REGION Network 65: Station 120 - Signalization (panel UH12)
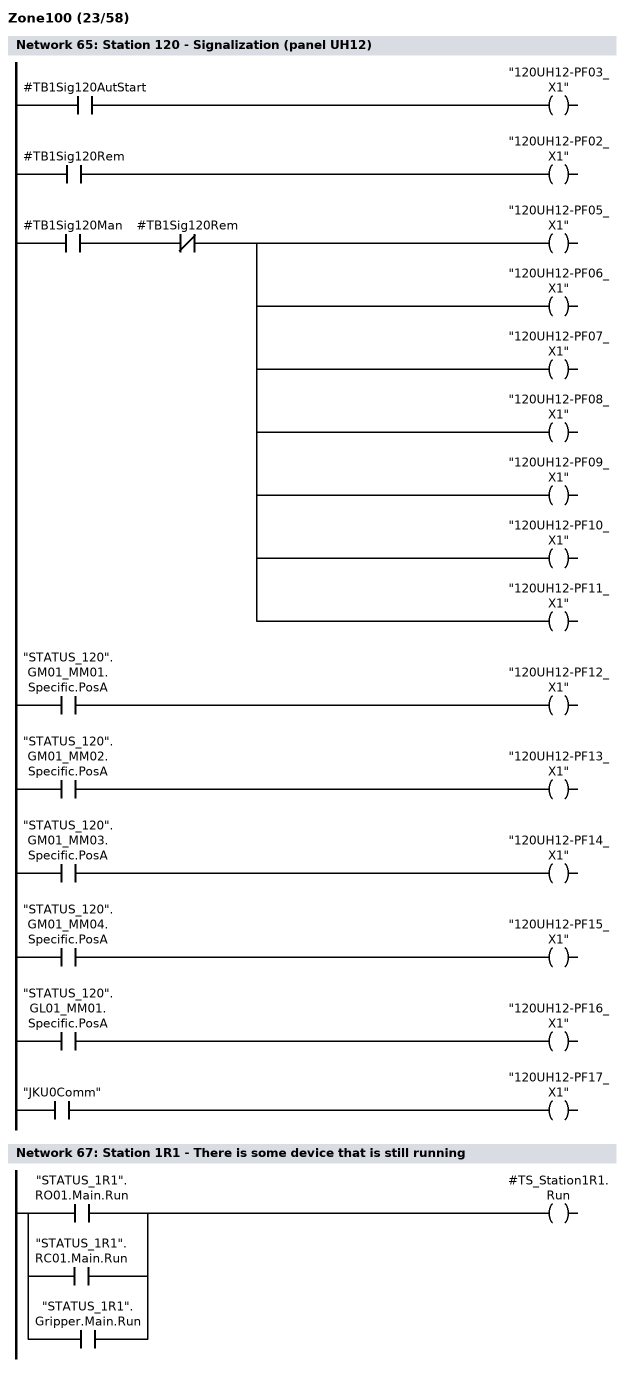
   RUNG wire#powerrail
      Contact( #TB1Sig120AutStart )
      Coil( "120UH12-PF03_X1" )
   END_RUNG
   RUNG wire#powerrail
      Contact( #TB1Sig120Rem )
      Coil( "120UH12-PF02_X1" )
   END_RUNG
   RUNG wire#powerrail
      Contact( #TB1Sig120Man )
      I_Contact( #TB1Sig120Rem )
      wire#w1
      Coil( "120UH12-PF05_X1" )
   END_RUNG
   RUNG wire#w1
      Coil( "120UH12-PF06_X1" )
   END_RUNG
   RUNG wire#w1
      Coil( "120UH12-PF07_X1" )
   END_RUNG
   RUNG wire#w1
      Coil( "120UH12-PF08_X1" )
   END_RUNG
   RUNG wire#w1
      Coil( "120UH12-PF09_X1" )
   END_RUNG
   RUNG wire#w1
      Coil( "120UH12-PF10_X1" )
   END_RUNG
   RUNG wire#w1
      Coil( "120UH12-PF11_X1" )
   END_RUNG
   RUNG wire#powerrail
      Contact( "STATUS_120".GM01_MM01.Specific.PosA )
      Coil( "120UH12-PF12_X1" )
   END_RUNG
   RUNG wire#powerrail
      Contact( "STATUS_120".GM01_MM02.Specific.PosA )
      Coil( "120UH12-PF13_X1" )
   END_RUNG
   RUNG wire#powerrail
      Contact( "STATUS_120".GM01_MM03.Specific.PosA )
      Coil( "120UH12-PF14_X1" )
   END_RUNG
   RUNG wire#powerrail
      Contact( "STATUS_120".GM01_MM04.Specific.PosA )
      Coil( "120UH12-PF15_X1" )
   END_RUNG
   RUNG wire#powerrail
      Contact( "STATUS_120".GL01_MM01.Specific.PosA )
      Coil( "120UH12-PF16_X1" )
   END_RUNG
   RUNG wire#powerrail
      Contact( "JKU0Comm" )
      Coil( "120UH12-PF17_X1" )
   END_RUNG
   // the same network as SCL:
   "120UH12-PF03_X1" := #TB1Sig120AutStart;
   "120UH12-PF02_X1" := #TB1Sig120Rem;
   "120UH12-PF05_X1" := #TB1Sig120Man AND NOT #TB1Sig120Rem;
   "120UH12-PF06_X1" := "120UH12-PF05_X1";
   "120UH12-PF07_X1" := "120UH12-PF05_X1";
   "120UH12-PF08_X1" := "120UH12-PF05_X1";
   "120UH12-PF09_X1" := "120UH12-PF05_X1";
   "120UH12-PF10_X1" := "120UH12-PF05_X1";
   "120UH12-PF11_X1" := "120UH12-PF05_X1";
   "120UH12-PF12_X1" := "STATUS_120".GM01_MM01.Specific.PosA;
   "120UH12-PF13_X1" := "STATUS_120".GM01_MM02.Specific.PosA;
   "120UH12-PF14_X1" := "STATUS_120".GM01_MM03.Specific.PosA;
   "120UH12-PF15_X1" := "STATUS_120".GM01_MM04.Specific.PosA;
   "120UH12-PF16_X1" := "STATUS_120".GL01_MM01.Specific.PosA;
   "120UH12-PF17_X1" := "JKU0Comm";
END_REGION

REGION Network 66: *************** Station 1R1 ***************
END_REGION

REGION Network 67: Station 1R1 - There is some device that is still running
   RUNG wire#powerrail
      Contact( "STATUS_1R1".RO01.Main.Run )
      wire#w1
      Coil( #TS_Station1R1.Run )
   END_RUNG
   RUNG wire#powerrail
      Contact( "STATUS_1R1".RC01.Main.Run )
   END_RUNG wire#w1
   RUNG wire#powerrail
      Contact( "STATUS_1R1".Gripper.Main.Run )
   END_RUNG wire#w1
   // the same network as SCL:
   #TS_Station1R1.Run := "STATUS_1R1".RO01.Main.Run OR "STATUS_1R1".RC01.Main.Run OR "STATUS_1R1".Gripper.Main.Run;
END_REGION

REGION Network 68: Station 1R1 - Warning
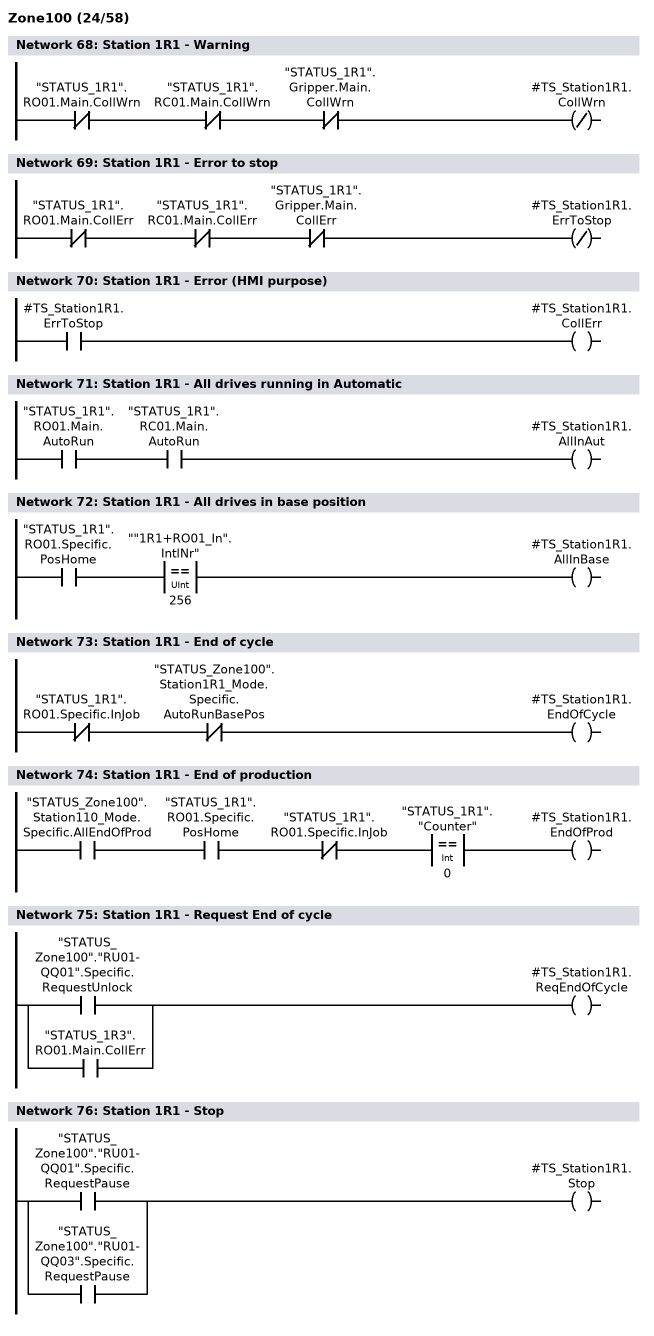
   RUNG wire#powerrail
      I_Contact( "STATUS_1R1".RO01.Main.CollWrn )
      I_Contact( "STATUS_1R1".RC01.Main.CollWrn )
      I_Contact( "STATUS_1R1".Gripper.Main.CollWrn )
      I_Coil( #TS_Station1R1.CollWrn )
   END_RUNG
   // the same network as SCL:
   #TS_Station1R1.CollWrn := NOT (NOT "STATUS_1R1".RO01.Main.CollWrn AND NOT "STATUS_1R1".RC01.Main.CollWrn AND NOT "STATUS_1R1".Gripper.Main.CollWrn);
END_REGION

REGION Network 69: Station 1R1 - Error to stop
   RUNG wire#powerrail
      I_Contact( "STATUS_1R1".RO01.Main.CollErr )
      I_Contact( "STATUS_1R1".RC01.Main.CollErr )
      I_Contact( "STATUS_1R1".Gripper.Main.CollErr )
      I_Coil( #TS_Station1R1.ErrToStop )
   END_RUNG
   // the same network as SCL:
   #TS_Station1R1.ErrToStop := NOT (NOT "STATUS_1R1".RO01.Main.CollErr AND NOT "STATUS_1R1".RC01.Main.CollErr AND NOT "STATUS_1R1".Gripper.Main.CollErr);
END_REGION

REGION Network 70: Station 1R1 - Error (HMI purpose)
   RUNG wire#powerrail
      Contact( #TS_Station1R1.ErrToStop )
      Coil( #TS_Station1R1.CollErr )
   END_RUNG
   // the same network as SCL:
   #TS_Station1R1.CollErr := #TS_Station1R1.ErrToStop;
END_REGION

REGION Network 71: Station 1R1 - All drives running in Automatic
   RUNG wire#powerrail
      Contact( "STATUS_1R1".RO01.Main.AutoRun )
      Contact( "STATUS_1R1".RC01.Main.AutoRun )
      Coil( #TS_Station1R1.AllInAut )
   END_RUNG
   // the same network as SCL:
   #TS_Station1R1.AllInAut := "STATUS_1R1".RO01.Main.AutoRun AND "STATUS_1R1".RC01.Main.AutoRun;
END_REGION

REGION Network 72: Station 1R1 - All drives in base position
   RUNG wire#powerrail
      Contact( "STATUS_1R1".RO01.Specific.PosHome )
      { S7_Templates := "SrcType := UInt" } EQ_Contact(in1 := ""1R1+RO01_In".IntlNr", in2 := 256)
      Coil( #TS_Station1R1.AllInBase )
   END_RUNG
   // the same network as SCL:
   // no checked SCL form for this network; see the picture
END_REGION

REGION Network 73: Station 1R1 - End of cycle
   RUNG wire#powerrail
      I_Contact( "STATUS_1R1".RO01.Specific.InJob )
      I_Contact( "STATUS_Zone100".Station1R1_Mode.Specific.AutoRunBasePos )
      Coil( #TS_Station1R1.EndOfCycle )
   END_RUNG
   // the same network as SCL:
   #TS_Station1R1.EndOfCycle := NOT "STATUS_1R1".RO01.Specific.InJob AND NOT "STATUS_Zone100".Station1R1_Mode.Specific.AutoRunBasePos;
END_REGION

REGION Network 74: Station 1R1 - End of production
   RUNG wire#powerrail
      Contact( "STATUS_Zone100".Station110_Mode.Specific.AllEndOfProd )
      Contact( "STATUS_1R1".RO01.Specific.PosHome )
      I_Contact( "STATUS_1R1".RO01.Specific.InJob )
      { S7_Templates := "SrcType := Int" } EQ_Contact(in1 := "STATUS_1R1"."Counter", in2 := 0)
      Coil( #TS_Station1R1.EndOfProd )
   END_RUNG
   // the same network as SCL:
   #TS_Station1R1.EndOfProd := "STATUS_Zone100".Station110_Mode.Specific.AllEndOfProd AND "STATUS_1R1".RO01.Specific.PosHome AND NOT "STATUS_1R1".RO01.Specific.InJob AND ("STATUS_1R1"."Counter" = 0);
END_REGION

REGION Network 75: Station 1R1 - Request End of cycle
   RUNG wire#powerrail
      Contact( "STATUS_Zone100"."RU01-QQ01".Specific.RequestUnlock )
      wire#w1
      Coil( #TS_Station1R1.ReqEndOfCycle )
   END_RUNG
   RUNG wire#powerrail
      Contact( "STATUS_1R3".RO01.Main.CollErr )
   END_RUNG wire#w1
   // the same network as SCL:
   #TS_Station1R1.ReqEndOfCycle := "STATUS_Zone100"."RU01-QQ01".Specific.RequestUnlock OR "STATUS_1R3".RO01.Main.CollErr;
END_REGION

REGION Network 76: Station 1R1 - Stop
   RUNG wire#powerrail
      Contact( "STATUS_Zone100"."RU01-QQ01".Specific.RequestPause )
      wire#w1
      Coil( #TS_Station1R1.Stop )
   END_RUNG
   RUNG wire#powerrail
      Contact( "STATUS_Zone100"."RU01-QQ03".Specific.RequestPause )
   END_RUNG wire#w1
   // the same network as SCL:
   #TS_Station1R1.Stop := "STATUS_Zone100"."RU01-QQ01".Specific.RequestPause OR "STATUS_Zone100"."RU01-QQ03".Specific.RequestPause;
END_REGION

REGION Network 77: Station 1R1 - Number of selected devices
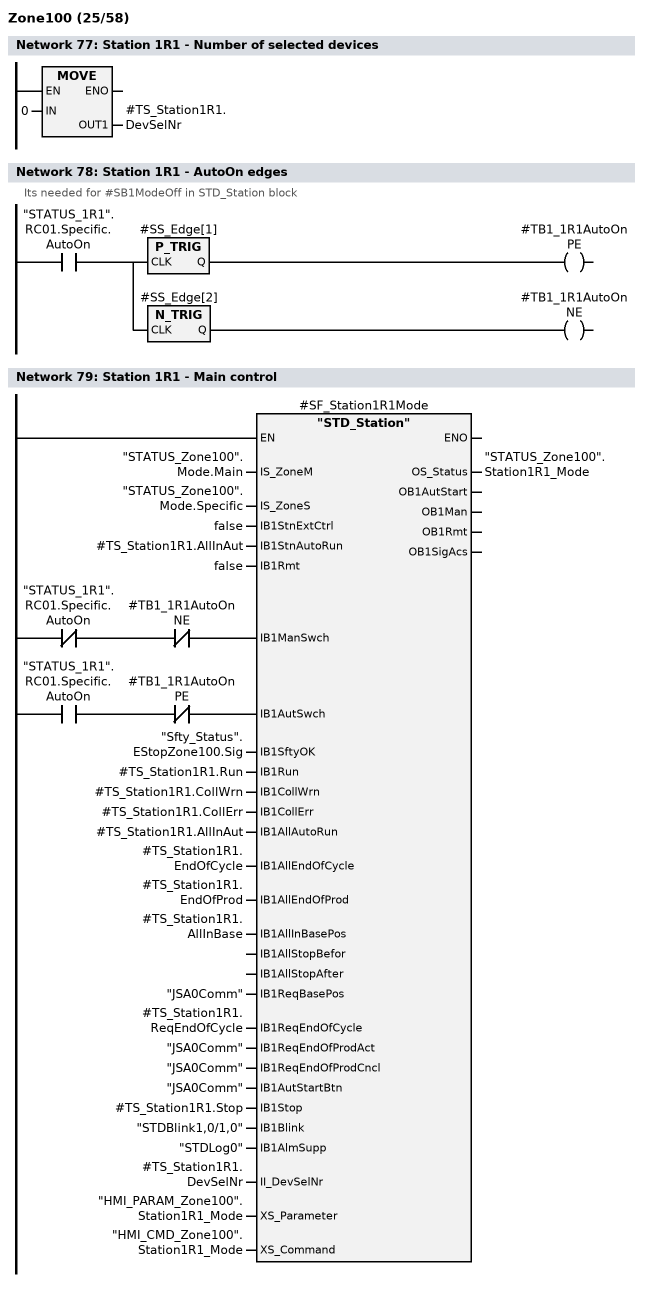
   RUNG wire#powerrail
      Move(in := 0, out1 => #TS_Station1R1.DevSelNr)
   END_RUNG
   // the same network as SCL:
   #TS_Station1R1.DevSelNr := 0;
END_REGION

REGION Network 78: Station 1R1 - AutoOn edges
   // Its needed for #SB1ModeOff in STD_Station block
   RUNG wire#powerrail
      Contact( "STATUS_1R1".RC01.Specific.AutoOn )
      wire#w1
      P_Trig( #SS_Edge[1] )
      Coil( #TB1_1R1AutoOnPE )
   END_RUNG
   RUNG wire#w1
      N_Trig( #SS_Edge[2] )
      Coil( #TB1_1R1AutoOnNE )
   END_RUNG
   // the same network as SCL:
   #_w1 := "STATUS_1R1".RC01.Specific.AutoOn AND NOT #SS_Edge[1];   // rising edge
   #SS_Edge[1] := "STATUS_1R1".RC01.Specific.AutoOn;
   #TB1_1R1AutoOnPE := #_w1;
   #_w2 := NOT "STATUS_1R1".RC01.Specific.AutoOn AND #SS_Edge[2];   // falling edge
   #SS_Edge[2] := "STATUS_1R1".RC01.Specific.AutoOn;
   #TB1_1R1AutoOnNE := #_w2;
END_REGION

REGION Network 79: Station 1R1 - Main control
   RUNG wire#powerrail
      #SF_Station1R1Mode(IB1ManSwch := wire#w1, IB1AutSwch := wire#w2, IS_ZoneM := "STATUS_Zone100".Mode.Main, IS_ZoneS := "STATUS_Zone100".Mode.Specific, IB1StnExtCtrl := false, IB1StnAutoRun := #TS_Station1R1.AllInAut, IB1Rmt := false, IB1SftyOK := "Sfty_Status".EStopZone100.Sig, IB1Run := #TS_Station1R1.Run, IB1CollWrn := #TS_Station1R1.CollWrn, IB1CollErr := #TS_Station1R1.CollErr, IB1AllAutoRun := #TS_Station1R1.AllInAut, IB1AllEndOfCycle := #TS_Station1R1.EndOfCycle, IB1AllEndOfProd := #TS_Station1R1.EndOfProd, IB1AllInBasePos := #TS_Station1R1.AllInBase, IB1AllStopBefor :=, IB1AllStopAfter :=, IB1ReqBasePos := "JSA0Comm", IB1ReqEndOfCycle := #TS_Station1R1.ReqEndOfCycle, IB1ReqEndOfProdAct := "JSA0Comm", IB1ReqEndOfProdCncl := "JSA0Comm", IB1AutStartBtn := "JSA0Comm", IB1Stop := #TS_Station1R1.Stop, IB1Blink := "STDBlink1,0/1,0", IB1AlmSupp := "STDLog0", II_DevSelNr := #TS_Station1R1.DevSelNr, XS_Parameter := "HMI_PARAM_Zone100".Station1R1_Mode, XS_Command := "HMI_CMD_Zone100".Station1R1_Mode, OS_Status => "STATUS_Zone100".Station1R1_Mode, OB1AutStart =>, OB1Man =>, OB1Rmt =>, OB1SigAcs =>)
   END_RUNG
   RUNG wire#powerrail
      I_Contact( "STATUS_1R1".RC01.Specific.AutoOn )
      I_Contact( #TB1_1R1AutoOnNE )
   END_RUNG wire#w1
   RUNG wire#powerrail
      Contact( "STATUS_1R1".RC01.Specific.AutoOn )
      I_Contact( #TB1_1R1AutoOnPE )
   END_RUNG wire#w2
   // the same network as SCL:
   #SF_Station1R1Mode(IS_ZoneM := "STATUS_Zone100".Mode.Main,   // "STD_Station"
                      IS_ZoneS := "STATUS_Zone100".Mode.Specific,
                      IB1StnExtCtrl := false,
                      IB1StnAutoRun := #TS_Station1R1.AllInAut,
                      IB1Rmt := false,
                      IB1ManSwch := NOT "STATUS_1R1".RC01.Specific.AutoOn AND NOT #TB1_1R1AutoOnNE,
                      IB1AutSwch := "STATUS_1R1".RC01.Specific.AutoOn AND NOT #TB1_1R1AutoOnPE,
                      IB1SftyOK := "Sfty_Status".EStopZone100.Sig,
                      IB1Run := #TS_Station1R1.Run,
                      IB1CollWrn := #TS_Station1R1.CollWrn,
                      IB1CollErr := #TS_Station1R1.CollErr,
                      IB1AllAutoRun := #TS_Station1R1.AllInAut,
                      IB1AllEndOfCycle := #TS_Station1R1.EndOfCycle,
                      IB1AllEndOfProd := #TS_Station1R1.EndOfProd,
                      IB1AllInBasePos := #TS_Station1R1.AllInBase,
                      IB1ReqBasePos := "JSA0Comm",
                      IB1ReqEndOfCycle := #TS_Station1R1.ReqEndOfCycle,
                      IB1ReqEndOfProdAct := "JSA0Comm",
                      IB1ReqEndOfProdCncl := "JSA0Comm",
                      IB1AutStartBtn := "JSA0Comm",
                      IB1Stop := #TS_Station1R1.Stop,
                      IB1Blink := "STDBlink1,0/1,0",
                      IB1AlmSupp := "STDLog0",
                      II_DevSelNr := #TS_Station1R1.DevSelNr,
                      XS_Parameter := "HMI_PARAM_Zone100".Station1R1_Mode,
                      XS_Command := "HMI_CMD_Zone100".Station1R1_Mode,
                      OS_Status => "STATUS_Zone100".Station1R1_Mode);
END_REGION

REGION Network 80: *************** Station 1R2 ***************
END_REGION

REGION Network 81: Station 1R2 - There is some device that is still running
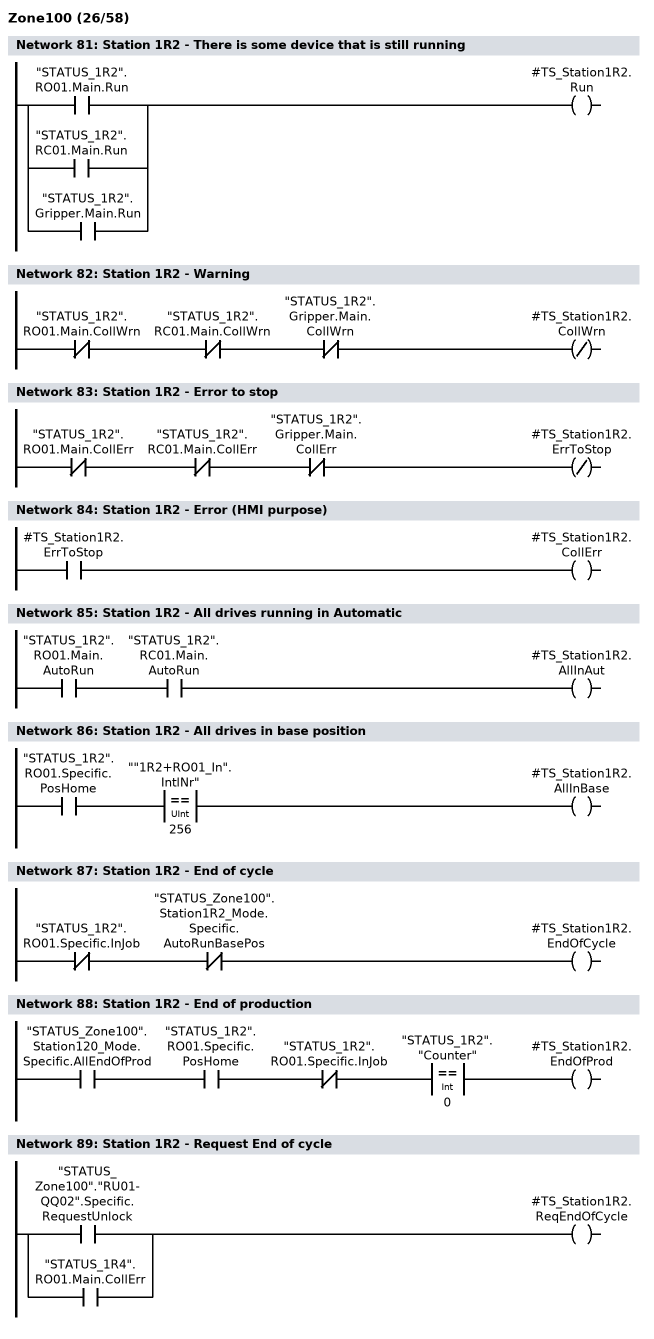
   RUNG wire#powerrail
      Contact( "STATUS_1R2".RO01.Main.Run )
      wire#w1
      Coil( #TS_Station1R2.Run )
   END_RUNG
   RUNG wire#powerrail
      Contact( "STATUS_1R2".RC01.Main.Run )
   END_RUNG wire#w1
   RUNG wire#powerrail
      Contact( "STATUS_1R2".Gripper.Main.Run )
   END_RUNG wire#w1
   // the same network as SCL:
   #TS_Station1R2.Run := "STATUS_1R2".RO01.Main.Run OR "STATUS_1R2".RC01.Main.Run OR "STATUS_1R2".Gripper.Main.Run;
END_REGION

REGION Network 82: Station 1R2 - Warning
   RUNG wire#powerrail
      I_Contact( "STATUS_1R2".RO01.Main.CollWrn )
      I_Contact( "STATUS_1R2".RC01.Main.CollWrn )
      I_Contact( "STATUS_1R2".Gripper.Main.CollWrn )
      I_Coil( #TS_Station1R2.CollWrn )
   END_RUNG
   // the same network as SCL:
   #TS_Station1R2.CollWrn := NOT (NOT "STATUS_1R2".RO01.Main.CollWrn AND NOT "STATUS_1R2".RC01.Main.CollWrn AND NOT "STATUS_1R2".Gripper.Main.CollWrn);
END_REGION

REGION Network 83: Station 1R2 - Error to stop
   RUNG wire#powerrail
      I_Contact( "STATUS_1R2".RO01.Main.CollErr )
      I_Contact( "STATUS_1R2".RC01.Main.CollErr )
      I_Contact( "STATUS_1R2".Gripper.Main.CollErr )
      I_Coil( #TS_Station1R2.ErrToStop )
   END_RUNG
   // the same network as SCL:
   #TS_Station1R2.ErrToStop := NOT (NOT "STATUS_1R2".RO01.Main.CollErr AND NOT "STATUS_1R2".RC01.Main.CollErr AND NOT "STATUS_1R2".Gripper.Main.CollErr);
END_REGION

REGION Network 84: Station 1R2 - Error (HMI purpose)
   RUNG wire#powerrail
      Contact( #TS_Station1R2.ErrToStop )
      Coil( #TS_Station1R2.CollErr )
   END_RUNG
   // the same network as SCL:
   #TS_Station1R2.CollErr := #TS_Station1R2.ErrToStop;
END_REGION

REGION Network 85: Station 1R2 - All drives running in Automatic
   RUNG wire#powerrail
      Contact( "STATUS_1R2".RO01.Main.AutoRun )
      Contact( "STATUS_1R2".RC01.Main.AutoRun )
      Coil( #TS_Station1R2.AllInAut )
   END_RUNG
   // the same network as SCL:
   #TS_Station1R2.AllInAut := "STATUS_1R2".RO01.Main.AutoRun AND "STATUS_1R2".RC01.Main.AutoRun;
END_REGION

REGION Network 86: Station 1R2 - All drives in base position
   RUNG wire#powerrail
      Contact( "STATUS_1R2".RO01.Specific.PosHome )
      { S7_Templates := "SrcType := UInt" } EQ_Contact(in1 := ""1R2+RO01_In".IntlNr", in2 := 256)
      Coil( #TS_Station1R2.AllInBase )
   END_RUNG
   // the same network as SCL:
   // no checked SCL form for this network; see the picture
END_REGION

REGION Network 87: Station 1R2 - End of cycle
   RUNG wire#powerrail
      I_Contact( "STATUS_1R2".RO01.Specific.InJob )
      I_Contact( "STATUS_Zone100".Station1R2_Mode.Specific.AutoRunBasePos )
      Coil( #TS_Station1R2.EndOfCycle )
   END_RUNG
   // the same network as SCL:
   #TS_Station1R2.EndOfCycle := NOT "STATUS_1R2".RO01.Specific.InJob AND NOT "STATUS_Zone100".Station1R2_Mode.Specific.AutoRunBasePos;
END_REGION

REGION Network 88: Station 1R2 - End of production
   RUNG wire#powerrail
      Contact( "STATUS_Zone100".Station120_Mode.Specific.AllEndOfProd )
      Contact( "STATUS_1R2".RO01.Specific.PosHome )
      I_Contact( "STATUS_1R2".RO01.Specific.InJob )
      { S7_Templates := "SrcType := Int" } EQ_Contact(in1 := "STATUS_1R2"."Counter", in2 := 0)
      Coil( #TS_Station1R2.EndOfProd )
   END_RUNG
   // the same network as SCL:
   #TS_Station1R2.EndOfProd := "STATUS_Zone100".Station120_Mode.Specific.AllEndOfProd AND "STATUS_1R2".RO01.Specific.PosHome AND NOT "STATUS_1R2".RO01.Specific.InJob AND ("STATUS_1R2"."Counter" = 0);
END_REGION

REGION Network 89: Station 1R2 - Request End of cycle
   RUNG wire#powerrail
      Contact( "STATUS_Zone100"."RU01-QQ02".Specific.RequestUnlock )
      wire#w1
      Coil( #TS_Station1R2.ReqEndOfCycle )
   END_RUNG
   RUNG wire#powerrail
      Contact( "STATUS_1R4".RO01.Main.CollErr )
   END_RUNG wire#w1
   // the same network as SCL:
   #TS_Station1R2.ReqEndOfCycle := "STATUS_Zone100"."RU01-QQ02".Specific.RequestUnlock OR "STATUS_1R4".RO01.Main.CollErr;
END_REGION

REGION Network 90: Station 1R2 - Stop
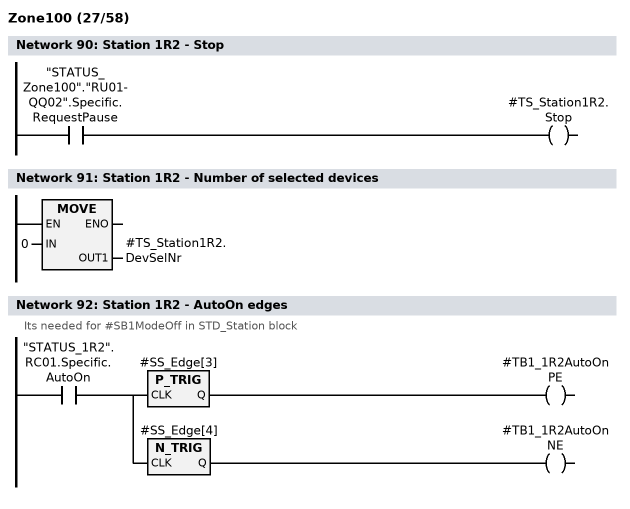
   RUNG wire#powerrail
      Contact( "STATUS_Zone100"."RU01-QQ02".Specific.RequestPause )
      Coil( #TS_Station1R2.Stop )
   END_RUNG
   // the same network as SCL:
   #TS_Station1R2.Stop := "STATUS_Zone100"."RU01-QQ02".Specific.RequestPause;
END_REGION

REGION Network 91: Station 1R2 - Number of selected devices
   RUNG wire#powerrail
      Move(in := 0, out1 => #TS_Station1R2.DevSelNr)
   END_RUNG
   // the same network as SCL:
   #TS_Station1R2.DevSelNr := 0;
END_REGION

REGION Network 92: Station 1R2 - AutoOn edges
   // Its needed for #SB1ModeOff in STD_Station block
   RUNG wire#powerrail
      Contact( "STATUS_1R2".RC01.Specific.AutoOn )
      wire#w1
      P_Trig( #SS_Edge[3] )
      Coil( #TB1_1R2AutoOnPE )
   END_RUNG
   RUNG wire#w1
      N_Trig( #SS_Edge[4] )
      Coil( #TB1_1R2AutoOnNE )
   END_RUNG
   // the same network as SCL:
   #_w1 := "STATUS_1R2".RC01.Specific.AutoOn AND NOT #SS_Edge[3];   // rising edge
   #SS_Edge[3] := "STATUS_1R2".RC01.Specific.AutoOn;
   #TB1_1R2AutoOnPE := #_w1;
   #_w2 := NOT "STATUS_1R2".RC01.Specific.AutoOn AND #SS_Edge[4];   // falling edge
   #SS_Edge[4] := "STATUS_1R2".RC01.Specific.AutoOn;
   #TB1_1R2AutoOnNE := #_w2;
END_REGION

REGION Network 93: Station 1R2 - Main control
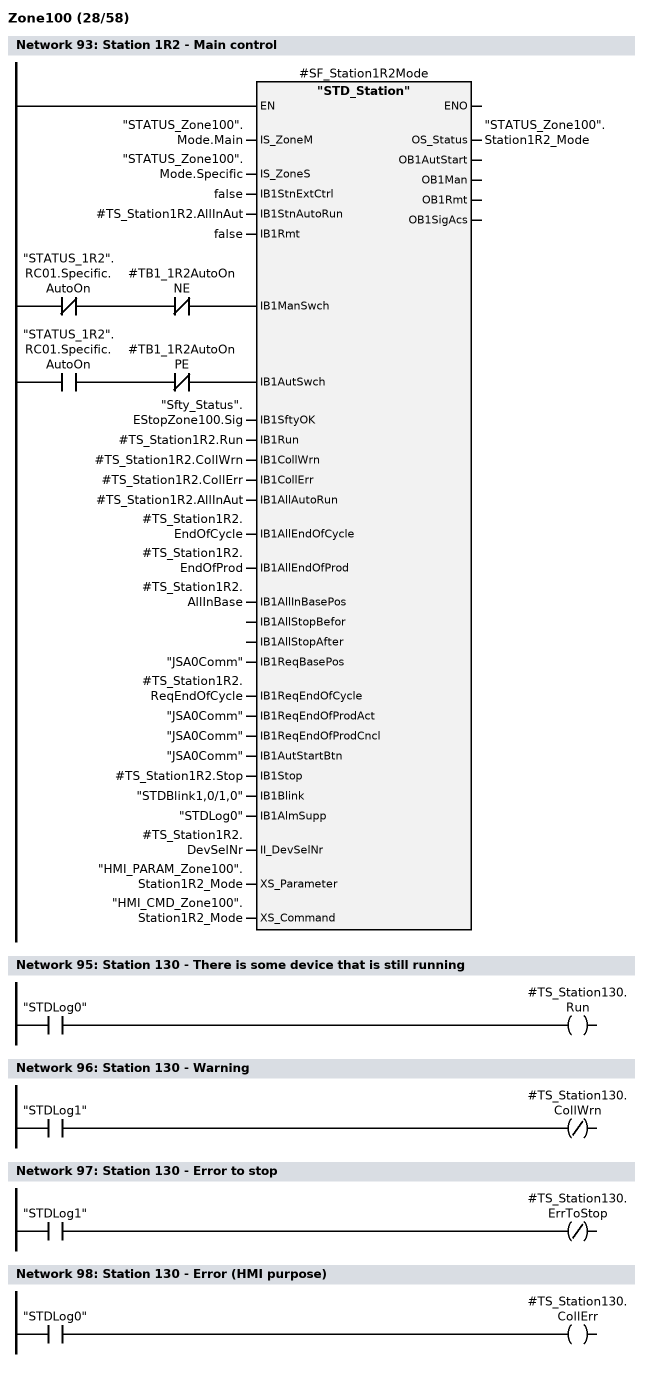
   RUNG wire#powerrail
      #SF_Station1R2Mode(IB1ManSwch := wire#w1, IB1AutSwch := wire#w2, IS_ZoneM := "STATUS_Zone100".Mode.Main, IS_ZoneS := "STATUS_Zone100".Mode.Specific, IB1StnExtCtrl := false, IB1StnAutoRun := #TS_Station1R2.AllInAut, IB1Rmt := false, IB1SftyOK := "Sfty_Status".EStopZone100.Sig, IB1Run := #TS_Station1R2.Run, IB1CollWrn := #TS_Station1R2.CollWrn, IB1CollErr := #TS_Station1R2.CollErr, IB1AllAutoRun := #TS_Station1R2.AllInAut, IB1AllEndOfCycle := #TS_Station1R2.EndOfCycle, IB1AllEndOfProd := #TS_Station1R2.EndOfProd, IB1AllInBasePos := #TS_Station1R2.AllInBase, IB1AllStopBefor :=, IB1AllStopAfter :=, IB1ReqBasePos := "JSA0Comm", IB1ReqEndOfCycle := #TS_Station1R2.ReqEndOfCycle, IB1ReqEndOfProdAct := "JSA0Comm", IB1ReqEndOfProdCncl := "JSA0Comm", IB1AutStartBtn := "JSA0Comm", IB1Stop := #TS_Station1R2.Stop, IB1Blink := "STDBlink1,0/1,0", IB1AlmSupp := "STDLog0", II_DevSelNr := #TS_Station1R2.DevSelNr, XS_Parameter := "HMI_PARAM_Zone100".Station1R2_Mode, XS_Command := "HMI_CMD_Zone100".Station1R2_Mode, OS_Status => "STATUS_Zone100".Station1R2_Mode, OB1AutStart =>, OB1Man =>, OB1Rmt =>, OB1SigAcs =>)
   END_RUNG
   RUNG wire#powerrail
      I_Contact( "STATUS_1R2".RC01.Specific.AutoOn )
      I_Contact( #TB1_1R2AutoOnNE )
   END_RUNG wire#w1
   RUNG wire#powerrail
      Contact( "STATUS_1R2".RC01.Specific.AutoOn )
      I_Contact( #TB1_1R2AutoOnPE )
   END_RUNG wire#w2
   // the same network as SCL:
   #SF_Station1R2Mode(IS_ZoneM := "STATUS_Zone100".Mode.Main,   // "STD_Station"
                      IS_ZoneS := "STATUS_Zone100".Mode.Specific,
                      IB1StnExtCtrl := false,
                      IB1StnAutoRun := #TS_Station1R2.AllInAut,
                      IB1Rmt := false,
                      IB1ManSwch := NOT "STATUS_1R2".RC01.Specific.AutoOn AND NOT #TB1_1R2AutoOnNE,
                      IB1AutSwch := "STATUS_1R2".RC01.Specific.AutoOn AND NOT #TB1_1R2AutoOnPE,
                      IB1SftyOK := "Sfty_Status".EStopZone100.Sig,
                      IB1Run := #TS_Station1R2.Run,
                      IB1CollWrn := #TS_Station1R2.CollWrn,
                      IB1CollErr := #TS_Station1R2.CollErr,
                      IB1AllAutoRun := #TS_Station1R2.AllInAut,
                      IB1AllEndOfCycle := #TS_Station1R2.EndOfCycle,
                      IB1AllEndOfProd := #TS_Station1R2.EndOfProd,
                      IB1AllInBasePos := #TS_Station1R2.AllInBase,
                      IB1ReqBasePos := "JSA0Comm",
                      IB1ReqEndOfCycle := #TS_Station1R2.ReqEndOfCycle,
                      IB1ReqEndOfProdAct := "JSA0Comm",
                      IB1ReqEndOfProdCncl := "JSA0Comm",
                      IB1AutStartBtn := "JSA0Comm",
                      IB1Stop := #TS_Station1R2.Stop,
                      IB1Blink := "STDBlink1,0/1,0",
                      IB1AlmSupp := "STDLog0",
                      II_DevSelNr := #TS_Station1R2.DevSelNr,
                      XS_Parameter := "HMI_PARAM_Zone100".Station1R2_Mode,
                      XS_Command := "HMI_CMD_Zone100".Station1R2_Mode,
                      OS_Status => "STATUS_Zone100".Station1R2_Mode);
END_REGION

REGION Network 94: *************** Station 130 ***************
END_REGION

REGION Network 95: Station 130 - There is some device that is still running
   RUNG wire#powerrail
      Contact( "STDLog0" )
      Coil( #TS_Station130.Run )
   END_RUNG
   // the same network as SCL:
   #TS_Station130.Run := "STDLog0";
END_REGION

REGION Network 96: Station 130 - Warning
   RUNG wire#powerrail
      Contact( "STDLog1" )
      I_Coil( #TS_Station130.CollWrn )
   END_RUNG
   // the same network as SCL:
   #TS_Station130.CollWrn := NOT "STDLog1";
END_REGION

REGION Network 97: Station 130 - Error to stop
   RUNG wire#powerrail
      Contact( "STDLog1" )
      I_Coil( #TS_Station130.ErrToStop )
   END_RUNG
   // the same network as SCL:
   #TS_Station130.ErrToStop := NOT "STDLog1";
END_REGION

REGION Network 98: Station 130 - Error (HMI purpose)
   RUNG wire#powerrail
      Contact( "STDLog0" )
      Coil( #TS_Station130.CollErr )
   END_RUNG
   // the same network as SCL:
   #TS_Station130.CollErr := "STDLog0";
END_REGION

REGION Network 99: Station 130 - All drives running in Automatic
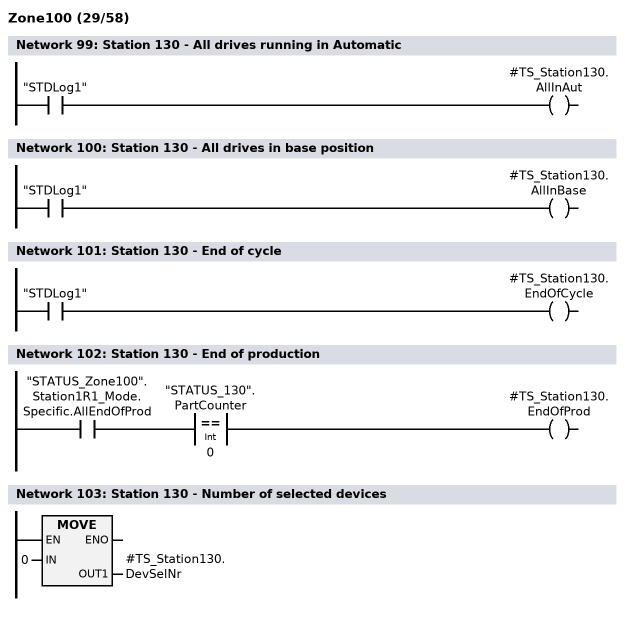
   RUNG wire#powerrail
      Contact( "STDLog1" )
      Coil( #TS_Station130.AllInAut )
   END_RUNG
   // the same network as SCL:
   #TS_Station130.AllInAut := "STDLog1";
END_REGION

REGION Network 100: Station 130 - All drives in base position
   RUNG wire#powerrail
      Contact( "STDLog1" )
      Coil( #TS_Station130.AllInBase )
   END_RUNG
   // the same network as SCL:
   #TS_Station130.AllInBase := "STDLog1";
END_REGION

REGION Network 101: Station 130 - End of cycle
   RUNG wire#powerrail
      Contact( "STDLog1" )
      Coil( #TS_Station130.EndOfCycle )
   END_RUNG
   // the same network as SCL:
   #TS_Station130.EndOfCycle := "STDLog1";
END_REGION

REGION Network 102: Station 130 - End of production
   RUNG wire#powerrail
      Contact( "STATUS_Zone100".Station1R1_Mode.Specific.AllEndOfProd )
      { S7_Templates := "SrcType := Int" } EQ_Contact(in1 := "STATUS_130".PartCounter, in2 := 0)
      Coil( #TS_Station130.EndOfProd )
   END_RUNG
   // the same network as SCL:
   #TS_Station130.EndOfProd := "STATUS_Zone100".Station1R1_Mode.Specific.AllEndOfProd AND ("STATUS_130".PartCounter = 0);
END_REGION

REGION Network 103: Station 130 - Number of selected devices
   RUNG wire#powerrail
      Move(in := 0, out1 => #TS_Station130.DevSelNr)
   END_RUNG
   // the same network as SCL:
   #TS_Station130.DevSelNr := 0;
END_REGION

REGION Network 104: Station 130 - Main control
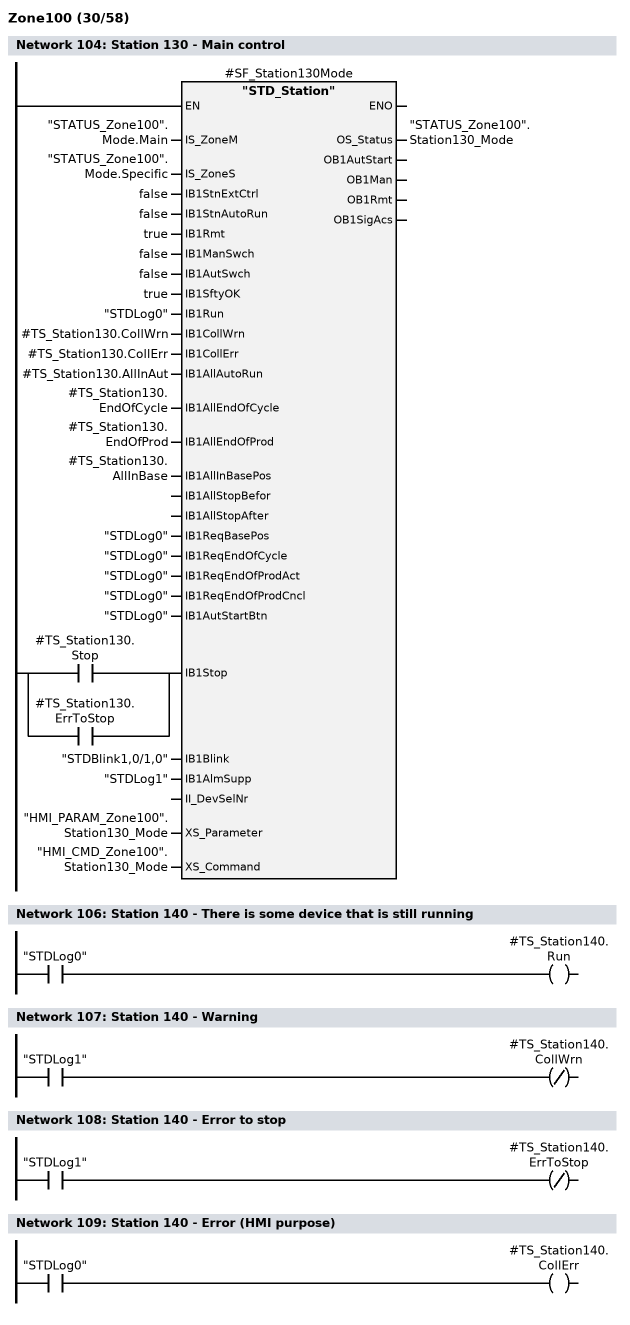
   RUNG wire#powerrail
      #SF_Station130Mode(IB1Stop := wire#w1, IS_ZoneM := "STATUS_Zone100".Mode.Main, IS_ZoneS := "STATUS_Zone100".Mode.Specific, IB1StnExtCtrl := false, IB1StnAutoRun := false, IB1Rmt := true, IB1ManSwch := false, IB1AutSwch := false, IB1SftyOK := true, IB1Run := "STDLog0", IB1CollWrn := #TS_Station130.CollWrn, IB1CollErr := #TS_Station130.CollErr, IB1AllAutoRun := #TS_Station130.AllInAut, IB1AllEndOfCycle := #TS_Station130.EndOfCycle, IB1AllEndOfProd := #TS_Station130.EndOfProd, IB1AllInBasePos := #TS_Station130.AllInBase, IB1AllStopBefor :=, IB1AllStopAfter :=, IB1ReqBasePos := "STDLog0", IB1ReqEndOfCycle := "STDLog0", IB1ReqEndOfProdAct := "STDLog0", IB1ReqEndOfProdCncl := "STDLog0", IB1AutStartBtn := "STDLog0", IB1Blink := "STDBlink1,0/1,0", IB1AlmSupp := "STDLog1", II_DevSelNr :=, XS_Parameter := "HMI_PARAM_Zone100".Station130_Mode, XS_Command := "HMI_CMD_Zone100".Station130_Mode, OS_Status => "STATUS_Zone100".Station130_Mode, OB1AutStart =>, OB1Man =>, OB1Rmt =>, OB1SigAcs =>)
   END_RUNG
   RUNG wire#powerrail
      Contact( #TS_Station130.Stop )
   END_RUNG wire#w1
   RUNG wire#powerrail
      Contact( #TS_Station130.ErrToStop )
   END_RUNG wire#w1
   // the same network as SCL:
   #SF_Station130Mode(IS_ZoneM := "STATUS_Zone100".Mode.Main,   // "STD_Station"
                      IS_ZoneS := "STATUS_Zone100".Mode.Specific,
                      IB1StnExtCtrl := false,
                      IB1StnAutoRun := false,
                      IB1Rmt := true,
                      IB1ManSwch := false,
                      IB1AutSwch := false,
                      IB1SftyOK := true,
                      IB1Run := "STDLog0",
                      IB1CollWrn := #TS_Station130.CollWrn,
                      IB1CollErr := #TS_Station130.CollErr,
                      IB1AllAutoRun := #TS_Station130.AllInAut,
                      IB1AllEndOfCycle := #TS_Station130.EndOfCycle,
                      IB1AllEndOfProd := #TS_Station130.EndOfProd,
                      IB1AllInBasePos := #TS_Station130.AllInBase,
                      IB1ReqBasePos := "STDLog0",
                      IB1ReqEndOfCycle := "STDLog0",
                      IB1ReqEndOfProdAct := "STDLog0",
                      IB1ReqEndOfProdCncl := "STDLog0",
                      IB1AutStartBtn := "STDLog0",
                      IB1Stop := #TS_Station130.Stop OR #TS_Station130.ErrToStop,
                      IB1Blink := "STDBlink1,0/1,0",
                      IB1AlmSupp := "STDLog1",
                      XS_Parameter := "HMI_PARAM_Zone100".Station130_Mode,
                      XS_Command := "HMI_CMD_Zone100".Station130_Mode,
                      OS_Status => "STATUS_Zone100".Station130_Mode);
END_REGION

REGION Network 105: *************** Station 140 ***************
END_REGION

REGION Network 106: Station 140 - There is some device that is still running
   RUNG wire#powerrail
      Contact( "STDLog0" )
      Coil( #TS_Station140.Run )
   END_RUNG
   // the same network as SCL:
   #TS_Station140.Run := "STDLog0";
END_REGION

REGION Network 107: Station 140 - Warning
   RUNG wire#powerrail
      Contact( "STDLog1" )
      I_Coil( #TS_Station140.CollWrn )
   END_RUNG
   // the same network as SCL:
   #TS_Station140.CollWrn := NOT "STDLog1";
END_REGION

REGION Network 108: Station 140 - Error to stop
   RUNG wire#powerrail
      Contact( "STDLog1" )
      I_Coil( #TS_Station140.ErrToStop )
   END_RUNG
   // the same network as SCL:
   #TS_Station140.ErrToStop := NOT "STDLog1";
END_REGION

REGION Network 109: Station 140 - Error (HMI purpose)
   RUNG wire#powerrail
      Contact( "STDLog0" )
      Coil( #TS_Station140.CollErr )
   END_RUNG
   // the same network as SCL:
   #TS_Station140.CollErr := "STDLog0";
END_REGION

REGION Network 110: Station 140 - All drives running in Automatic
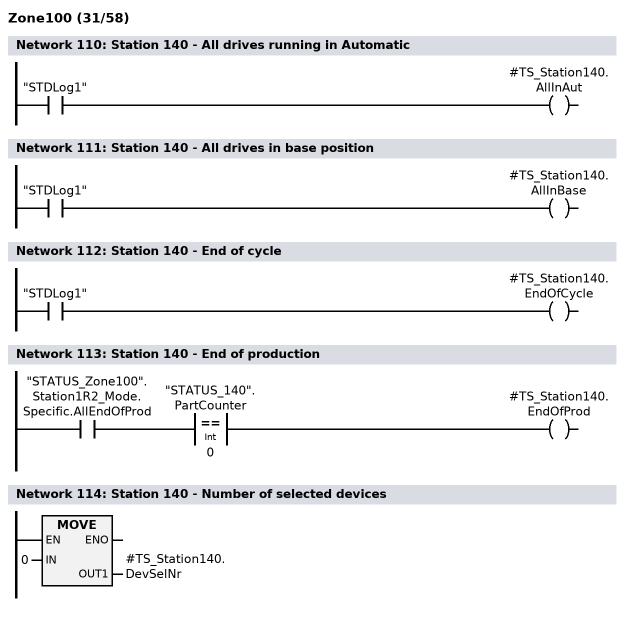
   RUNG wire#powerrail
      Contact( "STDLog1" )
      Coil( #TS_Station140.AllInAut )
   END_RUNG
   // the same network as SCL:
   #TS_Station140.AllInAut := "STDLog1";
END_REGION

REGION Network 111: Station 140 - All drives in base position
   RUNG wire#powerrail
      Contact( "STDLog1" )
      Coil( #TS_Station140.AllInBase )
   END_RUNG
   // the same network as SCL:
   #TS_Station140.AllInBase := "STDLog1";
END_REGION

REGION Network 112: Station 140 - End of cycle
   RUNG wire#powerrail
      Contact( "STDLog1" )
      Coil( #TS_Station140.EndOfCycle )
   END_RUNG
   // the same network as SCL:
   #TS_Station140.EndOfCycle := "STDLog1";
END_REGION

REGION Network 113: Station 140 - End of production
   RUNG wire#powerrail
      Contact( "STATUS_Zone100".Station1R2_Mode.Specific.AllEndOfProd )
      { S7_Templates := "SrcType := Int" } EQ_Contact(in1 := "STATUS_140".PartCounter, in2 := 0)
      Coil( #TS_Station140.EndOfProd )
   END_RUNG
   // the same network as SCL:
   #TS_Station140.EndOfProd := "STATUS_Zone100".Station1R2_Mode.Specific.AllEndOfProd AND ("STATUS_140".PartCounter = 0);
END_REGION

REGION Network 114: Station 140 - Number of selected devices
   RUNG wire#powerrail
      Move(in := 0, out1 => #TS_Station140.DevSelNr)
   END_RUNG
   // the same network as SCL:
   #TS_Station140.DevSelNr := 0;
END_REGION

REGION Network 115: Station 140 - Main control
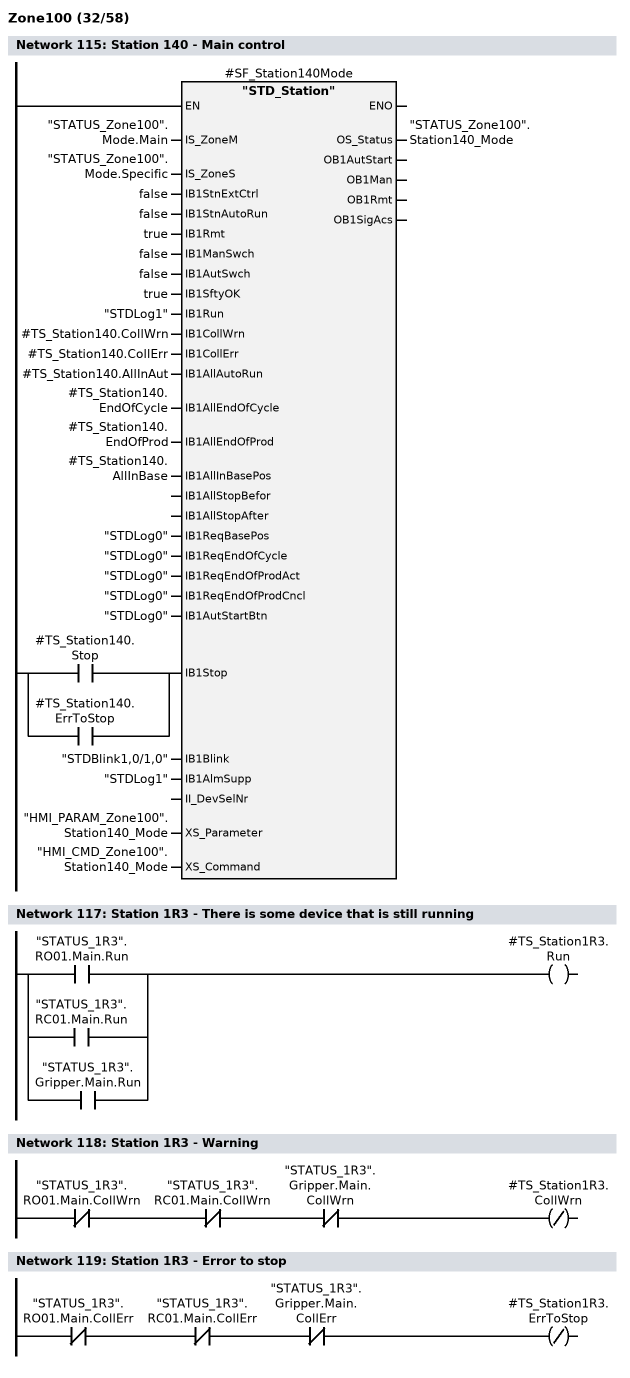
   RUNG wire#powerrail
      #SF_Station140Mode(IB1Stop := wire#w1, IS_ZoneM := "STATUS_Zone100".Mode.Main, IS_ZoneS := "STATUS_Zone100".Mode.Specific, IB1StnExtCtrl := false, IB1StnAutoRun := false, IB1Rmt := true, IB1ManSwch := false, IB1AutSwch := false, IB1SftyOK := true, IB1Run := "STDLog1", IB1CollWrn := #TS_Station140.CollWrn, IB1CollErr := #TS_Station140.CollErr, IB1AllAutoRun := #TS_Station140.AllInAut, IB1AllEndOfCycle := #TS_Station140.EndOfCycle, IB1AllEndOfProd := #TS_Station140.EndOfProd, IB1AllInBasePos := #TS_Station140.AllInBase, IB1AllStopBefor :=, IB1AllStopAfter :=, IB1ReqBasePos := "STDLog0", IB1ReqEndOfCycle := "STDLog0", IB1ReqEndOfProdAct := "STDLog0", IB1ReqEndOfProdCncl := "STDLog0", IB1AutStartBtn := "STDLog0", IB1Blink := "STDBlink1,0/1,0", IB1AlmSupp := "STDLog1", II_DevSelNr :=, XS_Parameter := "HMI_PARAM_Zone100".Station140_Mode, XS_Command := "HMI_CMD_Zone100".Station140_Mode, OS_Status => "STATUS_Zone100".Station140_Mode, OB1AutStart =>, OB1Man =>, OB1Rmt =>, OB1SigAcs =>)
   END_RUNG
   RUNG wire#powerrail
      Contact( #TS_Station140.Stop )
   END_RUNG wire#w1
   RUNG wire#powerrail
      Contact( #TS_Station140.ErrToStop )
   END_RUNG wire#w1
   // the same network as SCL:
   #SF_Station140Mode(IS_ZoneM := "STATUS_Zone100".Mode.Main,   // "STD_Station"
                      IS_ZoneS := "STATUS_Zone100".Mode.Specific,
                      IB1StnExtCtrl := false,
                      IB1StnAutoRun := false,
                      IB1Rmt := true,
                      IB1ManSwch := false,
                      IB1AutSwch := false,
                      IB1SftyOK := true,
                      IB1Run := "STDLog1",
                      IB1CollWrn := #TS_Station140.CollWrn,
                      IB1CollErr := #TS_Station140.CollErr,
                      IB1AllAutoRun := #TS_Station140.AllInAut,
                      IB1AllEndOfCycle := #TS_Station140.EndOfCycle,
                      IB1AllEndOfProd := #TS_Station140.EndOfProd,
                      IB1AllInBasePos := #TS_Station140.AllInBase,
                      IB1ReqBasePos := "STDLog0",
                      IB1ReqEndOfCycle := "STDLog0",
                      IB1ReqEndOfProdAct := "STDLog0",
                      IB1ReqEndOfProdCncl := "STDLog0",
                      IB1AutStartBtn := "STDLog0",
                      IB1Stop := #TS_Station140.Stop OR #TS_Station140.ErrToStop,
                      IB1Blink := "STDBlink1,0/1,0",
                      IB1AlmSupp := "STDLog1",
                      XS_Parameter := "HMI_PARAM_Zone100".Station140_Mode,
                      XS_Command := "HMI_CMD_Zone100".Station140_Mode,
                      OS_Status => "STATUS_Zone100".Station140_Mode);
END_REGION

REGION Network 116: *************** Station 1R3 ***************
END_REGION

REGION Network 117: Station 1R3 - There is some device that is still running
   RUNG wire#powerrail
      Contact( "STATUS_1R3".RO01.Main.Run )
      wire#w1
      Coil( #TS_Station1R3.Run )
   END_RUNG
   RUNG wire#powerrail
      Contact( "STATUS_1R3".RC01.Main.Run )
   END_RUNG wire#w1
   RUNG wire#powerrail
      Contact( "STATUS_1R3".Gripper.Main.Run )
   END_RUNG wire#w1
   // the same network as SCL:
   #TS_Station1R3.Run := "STATUS_1R3".RO01.Main.Run OR "STATUS_1R3".RC01.Main.Run OR "STATUS_1R3".Gripper.Main.Run;
END_REGION

REGION Network 118: Station 1R3 - Warning
   RUNG wire#powerrail
      I_Contact( "STATUS_1R3".RO01.Main.CollWrn )
      I_Contact( "STATUS_1R3".RC01.Main.CollWrn )
      I_Contact( "STATUS_1R3".Gripper.Main.CollWrn )
      I_Coil( #TS_Station1R3.CollWrn )
   END_RUNG
   // the same network as SCL:
   #TS_Station1R3.CollWrn := NOT (NOT "STATUS_1R3".RO01.Main.CollWrn AND NOT "STATUS_1R3".RC01.Main.CollWrn AND NOT "STATUS_1R3".Gripper.Main.CollWrn);
END_REGION

REGION Network 119: Station 1R3 - Error to stop
   RUNG wire#powerrail
      I_Contact( "STATUS_1R3".RO01.Main.CollErr )
      I_Contact( "STATUS_1R3".RC01.Main.CollErr )
      I_Contact( "STATUS_1R3".Gripper.Main.CollErr )
      I_Coil( #TS_Station1R3.ErrToStop )
   END_RUNG
   // the same network as SCL:
   #TS_Station1R3.ErrToStop := NOT (NOT "STATUS_1R3".RO01.Main.CollErr AND NOT "STATUS_1R3".RC01.Main.CollErr AND NOT "STATUS_1R3".Gripper.Main.CollErr);
END_REGION

REGION Network 120: Station 1R3 - Error (HMI purpose)
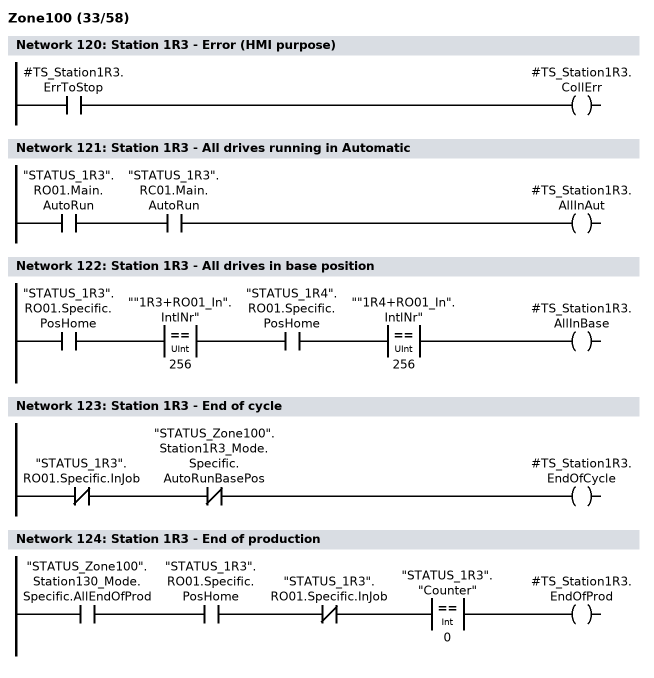
   RUNG wire#powerrail
      Contact( #TS_Station1R3.ErrToStop )
      Coil( #TS_Station1R3.CollErr )
   END_RUNG
   // the same network as SCL:
   #TS_Station1R3.CollErr := #TS_Station1R3.ErrToStop;
END_REGION

REGION Network 121: Station 1R3 - All drives running in Automatic
   RUNG wire#powerrail
      Contact( "STATUS_1R3".RO01.Main.AutoRun )
      Contact( "STATUS_1R3".RC01.Main.AutoRun )
      Coil( #TS_Station1R3.AllInAut )
   END_RUNG
   // the same network as SCL:
   #TS_Station1R3.AllInAut := "STATUS_1R3".RO01.Main.AutoRun AND "STATUS_1R3".RC01.Main.AutoRun;
END_REGION

REGION Network 122: Station 1R3 - All drives in base position
   RUNG wire#powerrail
      Contact( "STATUS_1R3".RO01.Specific.PosHome )
      { S7_Templates := "SrcType := UInt" } EQ_Contact(in1 := ""1R3+RO01_In".IntlNr", in2 := 256)
      Contact( "STATUS_1R4".RO01.Specific.PosHome )
      { S7_Templates := "SrcType := UInt" } EQ_Contact(in1 := ""1R4+RO01_In".IntlNr", in2 := 256)
      Coil( #TS_Station1R3.AllInBase )
   END_RUNG
   // the same network as SCL:
   // no checked SCL form for this network; see the picture
END_REGION

REGION Network 123: Station 1R3 - End of cycle
   RUNG wire#powerrail
      I_Contact( "STATUS_1R3".RO01.Specific.InJob )
      I_Contact( "STATUS_Zone100".Station1R3_Mode.Specific.AutoRunBasePos )
      Coil( #TS_Station1R3.EndOfCycle )
   END_RUNG
   // the same network as SCL:
   #TS_Station1R3.EndOfCycle := NOT "STATUS_1R3".RO01.Specific.InJob AND NOT "STATUS_Zone100".Station1R3_Mode.Specific.AutoRunBasePos;
END_REGION

REGION Network 124: Station 1R3 - End of production
   RUNG wire#powerrail
      Contact( "STATUS_Zone100".Station130_Mode.Specific.AllEndOfProd )
      Contact( "STATUS_1R3".RO01.Specific.PosHome )
      I_Contact( "STATUS_1R3".RO01.Specific.InJob )
      { S7_Templates := "SrcType := Int" } EQ_Contact(in1 := "STATUS_1R3"."Counter", in2 := 0)
      Coil( #TS_Station1R3.EndOfProd )
   END_RUNG
   // the same network as SCL:
   #TS_Station1R3.EndOfProd := "STATUS_Zone100".Station130_Mode.Specific.AllEndOfProd AND "STATUS_1R3".RO01.Specific.PosHome AND NOT "STATUS_1R3".RO01.Specific.InJob AND ("STATUS_1R3"."Counter" = 0);
END_REGION

REGION Network 125: Station 1R3 - Request End of cycle
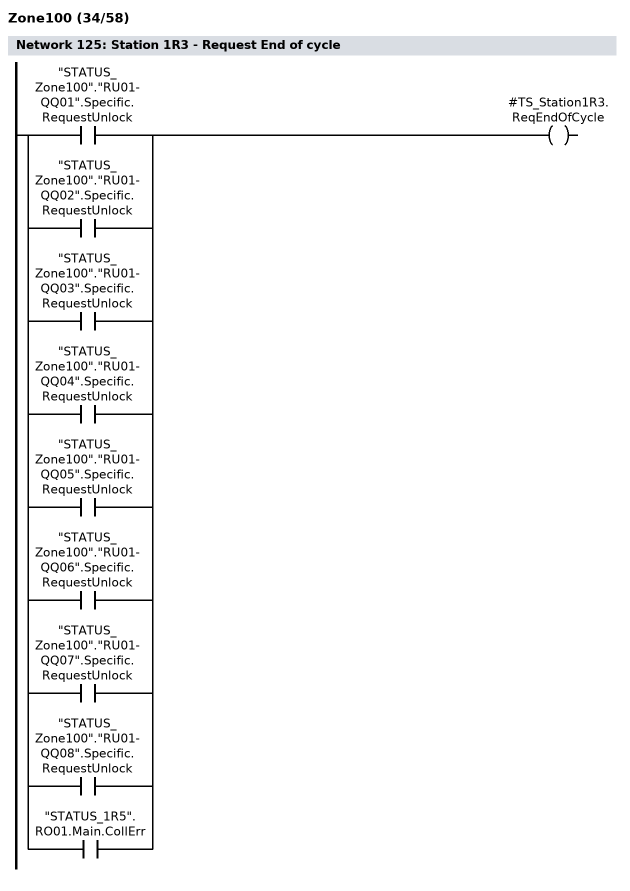
   RUNG wire#powerrail
      Contact( "STATUS_Zone100"."RU01-QQ01".Specific.RequestUnlock )
      wire#w1
      Coil( #TS_Station1R3.ReqEndOfCycle )
   END_RUNG
   RUNG wire#powerrail
      Contact( "STATUS_Zone100"."RU01-QQ02".Specific.RequestUnlock )
   END_RUNG wire#w1
   RUNG wire#powerrail
      Contact( "STATUS_Zone100"."RU01-QQ03".Specific.RequestUnlock )
   END_RUNG wire#w1
   RUNG wire#powerrail
      Contact( "STATUS_Zone100"."RU01-QQ04".Specific.RequestUnlock )
   END_RUNG wire#w1
   RUNG wire#powerrail
      Contact( "STATUS_Zone100"."RU01-QQ05".Specific.RequestUnlock )
   END_RUNG wire#w1
   RUNG wire#powerrail
      Contact( "STATUS_Zone100"."RU01-QQ06".Specific.RequestUnlock )
   END_RUNG wire#w1
   RUNG wire#powerrail
      Contact( "STATUS_Zone100"."RU01-QQ07".Specific.RequestUnlock )
   END_RUNG wire#w1
   RUNG wire#powerrail
      Contact( "STATUS_Zone100"."RU01-QQ08".Specific.RequestUnlock )
   END_RUNG wire#w1
   RUNG wire#powerrail
      Contact( "STATUS_1R5".RO01.Main.CollErr )
   END_RUNG wire#w1
   // the same network as SCL:
   #TS_Station1R3.ReqEndOfCycle := "STATUS_Zone100"."RU01-QQ01".Specific.RequestUnlock OR "STATUS_Zone100"."RU01-QQ02".Specific.RequestUnlock OR "STATUS_Zone100"."RU01-QQ03".Specific.RequestUnlock OR "STATUS_Zone100"."RU01-QQ04".Specific.RequestUnlock OR "STATUS_Zone100"."RU01-QQ05".Specific.RequestUnlock OR "STATUS_Zone100"."RU01-QQ06".Specific.RequestUnlock OR "STATUS_Zone100"."RU01-QQ07".Specific.RequestUnlock OR "STATUS_Zone100"."RU01-QQ08".Specific.RequestUnlock OR "STATUS_1R5".RO01.Main.CollErr;
END_REGION

REGION Network 126: Station 1R3 - Stop
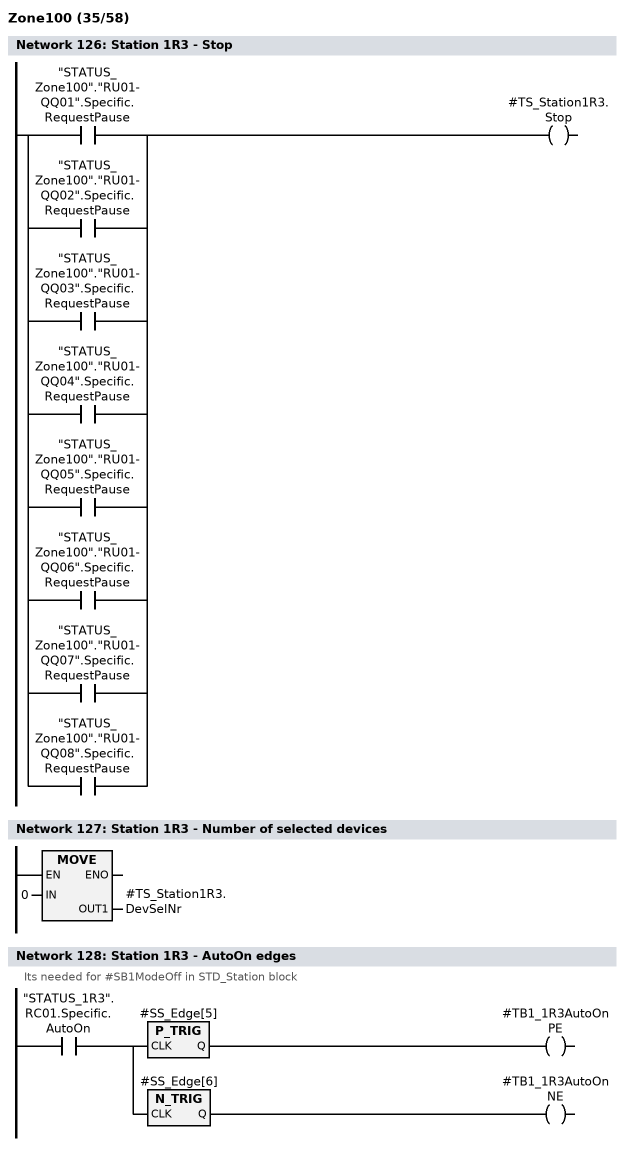
   RUNG wire#powerrail
      Contact( "STATUS_Zone100"."RU01-QQ01".Specific.RequestPause )
      wire#w1
      Coil( #TS_Station1R3.Stop )
   END_RUNG
   RUNG wire#powerrail
      Contact( "STATUS_Zone100"."RU01-QQ02".Specific.RequestPause )
   END_RUNG wire#w1
   RUNG wire#powerrail
      Contact( "STATUS_Zone100"."RU01-QQ03".Specific.RequestPause )
   END_RUNG wire#w1
   RUNG wire#powerrail
      Contact( "STATUS_Zone100"."RU01-QQ04".Specific.RequestPause )
   END_RUNG wire#w1
   RUNG wire#powerrail
      Contact( "STATUS_Zone100"."RU01-QQ05".Specific.RequestPause )
   END_RUNG wire#w1
   RUNG wire#powerrail
      Contact( "STATUS_Zone100"."RU01-QQ06".Specific.RequestPause )
   END_RUNG wire#w1
   RUNG wire#powerrail
      Contact( "STATUS_Zone100"."RU01-QQ07".Specific.RequestPause )
   END_RUNG wire#w1
   RUNG wire#powerrail
      Contact( "STATUS_Zone100"."RU01-QQ08".Specific.RequestPause )
   END_RUNG wire#w1
   // the same network as SCL:
   #TS_Station1R3.Stop := "STATUS_Zone100"."RU01-QQ01".Specific.RequestPause OR "STATUS_Zone100"."RU01-QQ02".Specific.RequestPause OR "STATUS_Zone100"."RU01-QQ03".Specific.RequestPause OR "STATUS_Zone100"."RU01-QQ04".Specific.RequestPause OR "STATUS_Zone100"."RU01-QQ05".Specific.RequestPause OR "STATUS_Zone100"."RU01-QQ06".Specific.RequestPause OR "STATUS_Zone100"."RU01-QQ07".Specific.RequestPause OR "STATUS_Zone100"."RU01-QQ08".Specific.RequestPause;
END_REGION

REGION Network 127: Station 1R3 - Number of selected devices
   RUNG wire#powerrail
      Move(in := 0, out1 => #TS_Station1R3.DevSelNr)
   END_RUNG
   // the same network as SCL:
   #TS_Station1R3.DevSelNr := 0;
END_REGION

REGION Network 128: Station 1R3 - AutoOn edges
   // Its needed for #SB1ModeOff in STD_Station block
   RUNG wire#powerrail
      Contact( "STATUS_1R3".RC01.Specific.AutoOn )
      wire#w1
      P_Trig( #SS_Edge[5] )
      Coil( #TB1_1R3AutoOnPE )
   END_RUNG
   RUNG wire#w1
      N_Trig( #SS_Edge[6] )
      Coil( #TB1_1R3AutoOnNE )
   END_RUNG
   // the same network as SCL:
   #_w1 := "STATUS_1R3".RC01.Specific.AutoOn AND NOT #SS_Edge[5];   // rising edge
   #SS_Edge[5] := "STATUS_1R3".RC01.Specific.AutoOn;
   #TB1_1R3AutoOnPE := #_w1;
   #_w2 := NOT "STATUS_1R3".RC01.Specific.AutoOn AND #SS_Edge[6];   // falling edge
   #SS_Edge[6] := "STATUS_1R3".RC01.Specific.AutoOn;
   #TB1_1R3AutoOnNE := #_w2;
END_REGION

REGION Network 129: Station 1R3 - Main control
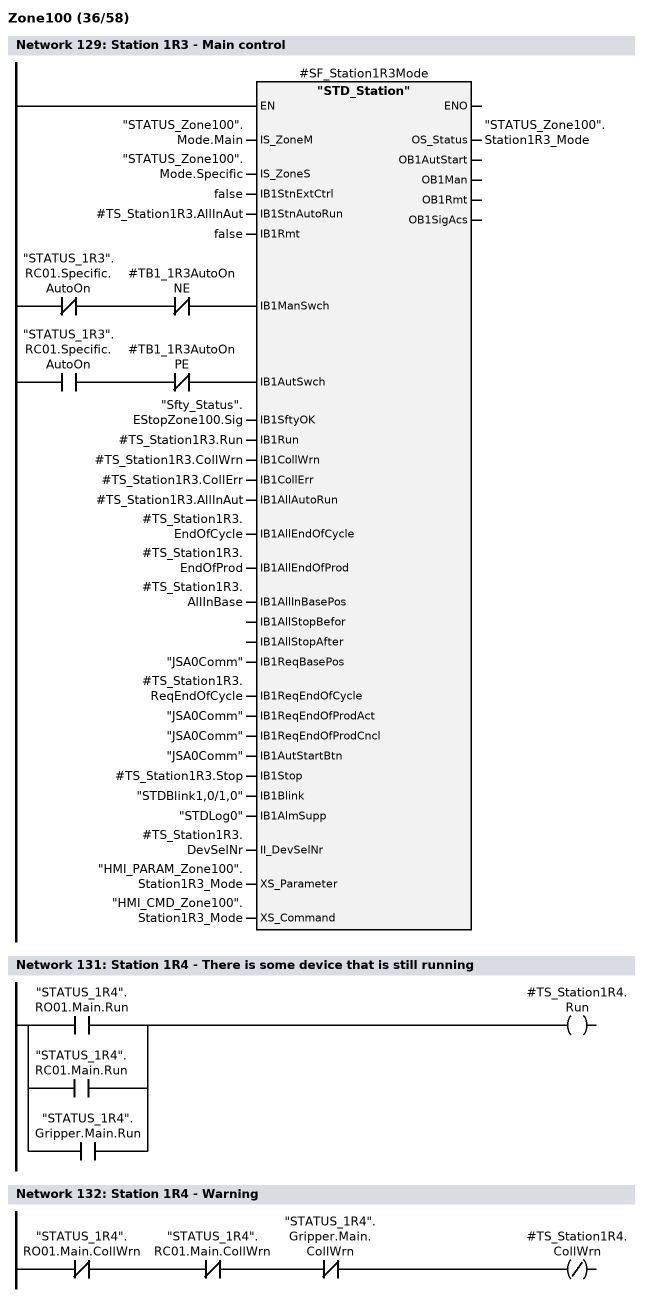
   RUNG wire#powerrail
      #SF_Station1R3Mode(IB1ManSwch := wire#w1, IB1AutSwch := wire#w2, IS_ZoneM := "STATUS_Zone100".Mode.Main, IS_ZoneS := "STATUS_Zone100".Mode.Specific, IB1StnExtCtrl := false, IB1StnAutoRun := #TS_Station1R3.AllInAut, IB1Rmt := false, IB1SftyOK := "Sfty_Status".EStopZone100.Sig, IB1Run := #TS_Station1R3.Run, IB1CollWrn := #TS_Station1R3.CollWrn, IB1CollErr := #TS_Station1R3.CollErr, IB1AllAutoRun := #TS_Station1R3.AllInAut, IB1AllEndOfCycle := #TS_Station1R3.EndOfCycle, IB1AllEndOfProd := #TS_Station1R3.EndOfProd, IB1AllInBasePos := #TS_Station1R3.AllInBase, IB1AllStopBefor :=, IB1AllStopAfter :=, IB1ReqBasePos := "JSA0Comm", IB1ReqEndOfCycle := #TS_Station1R3.ReqEndOfCycle, IB1ReqEndOfProdAct := "JSA0Comm", IB1ReqEndOfProdCncl := "JSA0Comm", IB1AutStartBtn := "JSA0Comm", IB1Stop := #TS_Station1R3.Stop, IB1Blink := "STDBlink1,0/1,0", IB1AlmSupp := "STDLog0", II_DevSelNr := #TS_Station1R3.DevSelNr, XS_Parameter := "HMI_PARAM_Zone100".Station1R3_Mode, XS_Command := "HMI_CMD_Zone100".Station1R3_Mode, OS_Status => "STATUS_Zone100".Station1R3_Mode, OB1AutStart =>, OB1Man =>, OB1Rmt =>, OB1SigAcs =>)
   END_RUNG
   RUNG wire#powerrail
      I_Contact( "STATUS_1R3".RC01.Specific.AutoOn )
      I_Contact( #TB1_1R3AutoOnNE )
   END_RUNG wire#w1
   RUNG wire#powerrail
      Contact( "STATUS_1R3".RC01.Specific.AutoOn )
      I_Contact( #TB1_1R3AutoOnPE )
   END_RUNG wire#w2
   // the same network as SCL:
   #SF_Station1R3Mode(IS_ZoneM := "STATUS_Zone100".Mode.Main,   // "STD_Station"
                      IS_ZoneS := "STATUS_Zone100".Mode.Specific,
                      IB1StnExtCtrl := false,
                      IB1StnAutoRun := #TS_Station1R3.AllInAut,
                      IB1Rmt := false,
                      IB1ManSwch := NOT "STATUS_1R3".RC01.Specific.AutoOn AND NOT #TB1_1R3AutoOnNE,
                      IB1AutSwch := "STATUS_1R3".RC01.Specific.AutoOn AND NOT #TB1_1R3AutoOnPE,
                      IB1SftyOK := "Sfty_Status".EStopZone100.Sig,
                      IB1Run := #TS_Station1R3.Run,
                      IB1CollWrn := #TS_Station1R3.CollWrn,
                      IB1CollErr := #TS_Station1R3.CollErr,
                      IB1AllAutoRun := #TS_Station1R3.AllInAut,
                      IB1AllEndOfCycle := #TS_Station1R3.EndOfCycle,
                      IB1AllEndOfProd := #TS_Station1R3.EndOfProd,
                      IB1AllInBasePos := #TS_Station1R3.AllInBase,
                      IB1ReqBasePos := "JSA0Comm",
                      IB1ReqEndOfCycle := #TS_Station1R3.ReqEndOfCycle,
                      IB1ReqEndOfProdAct := "JSA0Comm",
                      IB1ReqEndOfProdCncl := "JSA0Comm",
                      IB1AutStartBtn := "JSA0Comm",
                      IB1Stop := #TS_Station1R3.Stop,
                      IB1Blink := "STDBlink1,0/1,0",
                      IB1AlmSupp := "STDLog0",
                      II_DevSelNr := #TS_Station1R3.DevSelNr,
                      XS_Parameter := "HMI_PARAM_Zone100".Station1R3_Mode,
                      XS_Command := "HMI_CMD_Zone100".Station1R3_Mode,
                      OS_Status => "STATUS_Zone100".Station1R3_Mode);
END_REGION

REGION Network 130: *************** Station 1R4 ***************
END_REGION

REGION Network 131: Station 1R4 - There is some device that is still running
   RUNG wire#powerrail
      Contact( "STATUS_1R4".RO01.Main.Run )
      wire#w1
      Coil( #TS_Station1R4.Run )
   END_RUNG
   RUNG wire#powerrail
      Contact( "STATUS_1R4".RC01.Main.Run )
   END_RUNG wire#w1
   RUNG wire#powerrail
      Contact( "STATUS_1R4".Gripper.Main.Run )
   END_RUNG wire#w1
   // the same network as SCL:
   #TS_Station1R4.Run := "STATUS_1R4".RO01.Main.Run OR "STATUS_1R4".RC01.Main.Run OR "STATUS_1R4".Gripper.Main.Run;
END_REGION

REGION Network 132: Station 1R4 - Warning
   RUNG wire#powerrail
      I_Contact( "STATUS_1R4".RO01.Main.CollWrn )
      I_Contact( "STATUS_1R4".RC01.Main.CollWrn )
      I_Contact( "STATUS_1R4".Gripper.Main.CollWrn )
      I_Coil( #TS_Station1R4.CollWrn )
   END_RUNG
   // the same network as SCL:
   #TS_Station1R4.CollWrn := NOT (NOT "STATUS_1R4".RO01.Main.CollWrn AND NOT "STATUS_1R4".RC01.Main.CollWrn AND NOT "STATUS_1R4".Gripper.Main.CollWrn);
END_REGION

REGION Network 133: Station 1R4 - Error to stop
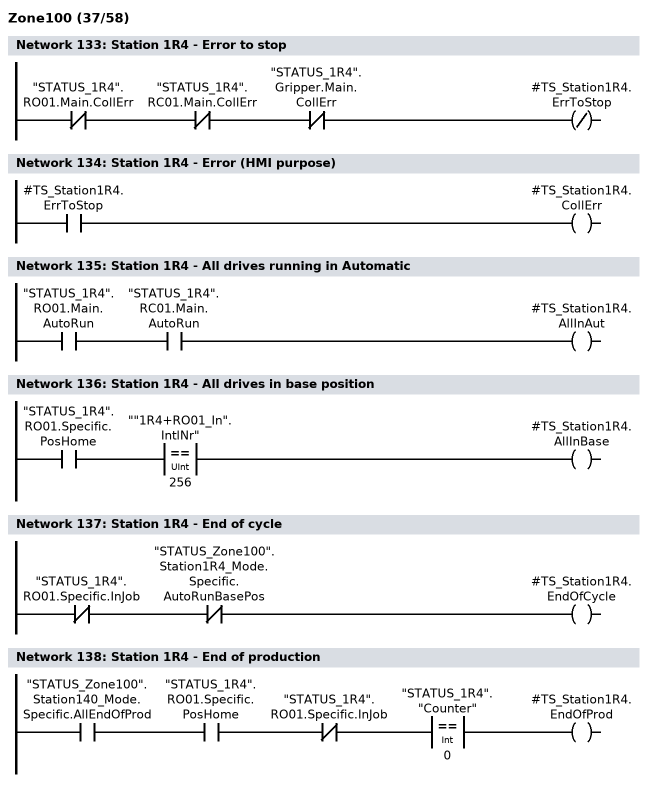
   RUNG wire#powerrail
      I_Contact( "STATUS_1R4".RO01.Main.CollErr )
      I_Contact( "STATUS_1R4".RC01.Main.CollErr )
      I_Contact( "STATUS_1R4".Gripper.Main.CollErr )
      I_Coil( #TS_Station1R4.ErrToStop )
   END_RUNG
   // the same network as SCL:
   #TS_Station1R4.ErrToStop := NOT (NOT "STATUS_1R4".RO01.Main.CollErr AND NOT "STATUS_1R4".RC01.Main.CollErr AND NOT "STATUS_1R4".Gripper.Main.CollErr);
END_REGION

REGION Network 134: Station 1R4 - Error (HMI purpose)
   RUNG wire#powerrail
      Contact( #TS_Station1R4.ErrToStop )
      Coil( #TS_Station1R4.CollErr )
   END_RUNG
   // the same network as SCL:
   #TS_Station1R4.CollErr := #TS_Station1R4.ErrToStop;
END_REGION

REGION Network 135: Station 1R4 - All drives running in Automatic
   RUNG wire#powerrail
      Contact( "STATUS_1R4".RO01.Main.AutoRun )
      Contact( "STATUS_1R4".RC01.Main.AutoRun )
      Coil( #TS_Station1R4.AllInAut )
   END_RUNG
   // the same network as SCL:
   #TS_Station1R4.AllInAut := "STATUS_1R4".RO01.Main.AutoRun AND "STATUS_1R4".RC01.Main.AutoRun;
END_REGION

REGION Network 136: Station 1R4 - All drives in base position
   RUNG wire#powerrail
      Contact( "STATUS_1R4".RO01.Specific.PosHome )
      { S7_Templates := "SrcType := UInt" } EQ_Contact(in1 := ""1R4+RO01_In".IntlNr", in2 := 256)
      Coil( #TS_Station1R4.AllInBase )
   END_RUNG
   // the same network as SCL:
   // no checked SCL form for this network; see the picture
END_REGION

REGION Network 137: Station 1R4 - End of cycle
   RUNG wire#powerrail
      I_Contact( "STATUS_1R4".RO01.Specific.InJob )
      I_Contact( "STATUS_Zone100".Station1R4_Mode.Specific.AutoRunBasePos )
      Coil( #TS_Station1R4.EndOfCycle )
   END_RUNG
   // the same network as SCL:
   #TS_Station1R4.EndOfCycle := NOT "STATUS_1R4".RO01.Specific.InJob AND NOT "STATUS_Zone100".Station1R4_Mode.Specific.AutoRunBasePos;
END_REGION

REGION Network 138: Station 1R4 - End of production
   RUNG wire#powerrail
      Contact( "STATUS_Zone100".Station140_Mode.Specific.AllEndOfProd )
      Contact( "STATUS_1R4".RO01.Specific.PosHome )
      I_Contact( "STATUS_1R4".RO01.Specific.InJob )
      { S7_Templates := "SrcType := Int" } EQ_Contact(in1 := "STATUS_1R4"."Counter", in2 := 0)
      Coil( #TS_Station1R4.EndOfProd )
   END_RUNG
   // the same network as SCL:
   #TS_Station1R4.EndOfProd := "STATUS_Zone100".Station140_Mode.Specific.AllEndOfProd AND "STATUS_1R4".RO01.Specific.PosHome AND NOT "STATUS_1R4".RO01.Specific.InJob AND ("STATUS_1R4"."Counter" = 0);
END_REGION

REGION Network 139: Station 1R4 - Request End of cycle
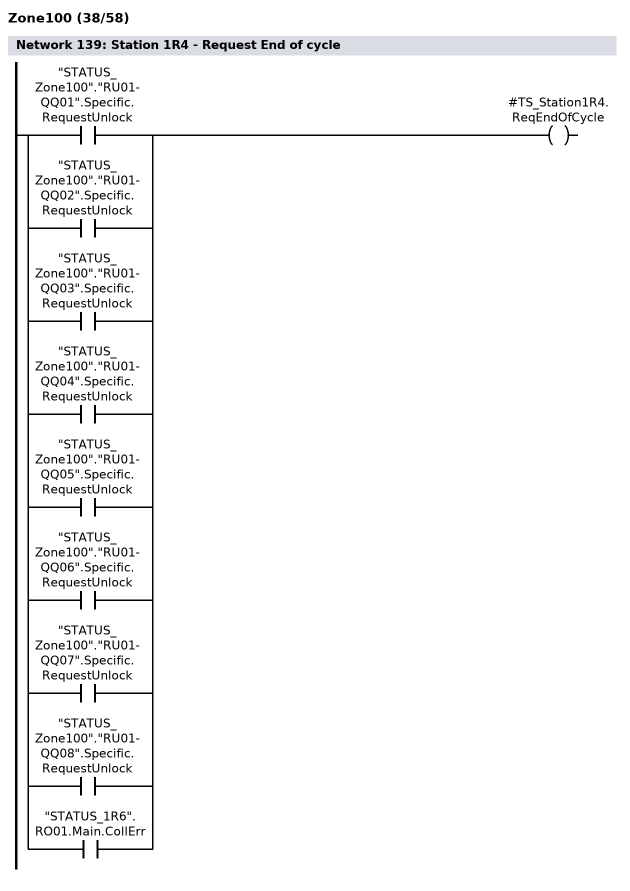
   RUNG wire#powerrail
      Contact( "STATUS_Zone100"."RU01-QQ01".Specific.RequestUnlock )
      wire#w1
      Coil( #TS_Station1R4.ReqEndOfCycle )
   END_RUNG
   RUNG wire#powerrail
      Contact( "STATUS_Zone100"."RU01-QQ02".Specific.RequestUnlock )
   END_RUNG wire#w1
   RUNG wire#powerrail
      Contact( "STATUS_Zone100"."RU01-QQ03".Specific.RequestUnlock )
   END_RUNG wire#w1
   RUNG wire#powerrail
      Contact( "STATUS_Zone100"."RU01-QQ04".Specific.RequestUnlock )
   END_RUNG wire#w1
   RUNG wire#powerrail
      Contact( "STATUS_Zone100"."RU01-QQ05".Specific.RequestUnlock )
   END_RUNG wire#w1
   RUNG wire#powerrail
      Contact( "STATUS_Zone100"."RU01-QQ06".Specific.RequestUnlock )
   END_RUNG wire#w1
   RUNG wire#powerrail
      Contact( "STATUS_Zone100"."RU01-QQ07".Specific.RequestUnlock )
   END_RUNG wire#w1
   RUNG wire#powerrail
      Contact( "STATUS_Zone100"."RU01-QQ08".Specific.RequestUnlock )
   END_RUNG wire#w1
   RUNG wire#powerrail
      Contact( "STATUS_1R6".RO01.Main.CollErr )
   END_RUNG wire#w1
   // the same network as SCL:
   #TS_Station1R4.ReqEndOfCycle := "STATUS_Zone100"."RU01-QQ01".Specific.RequestUnlock OR "STATUS_Zone100"."RU01-QQ02".Specific.RequestUnlock OR "STATUS_Zone100"."RU01-QQ03".Specific.RequestUnlock OR "STATUS_Zone100"."RU01-QQ04".Specific.RequestUnlock OR "STATUS_Zone100"."RU01-QQ05".Specific.RequestUnlock OR "STATUS_Zone100"."RU01-QQ06".Specific.RequestUnlock OR "STATUS_Zone100"."RU01-QQ07".Specific.RequestUnlock OR "STATUS_Zone100"."RU01-QQ08".Specific.RequestUnlock OR "STATUS_1R6".RO01.Main.CollErr;
END_REGION

REGION Network 140: Station 1R4 - Stop
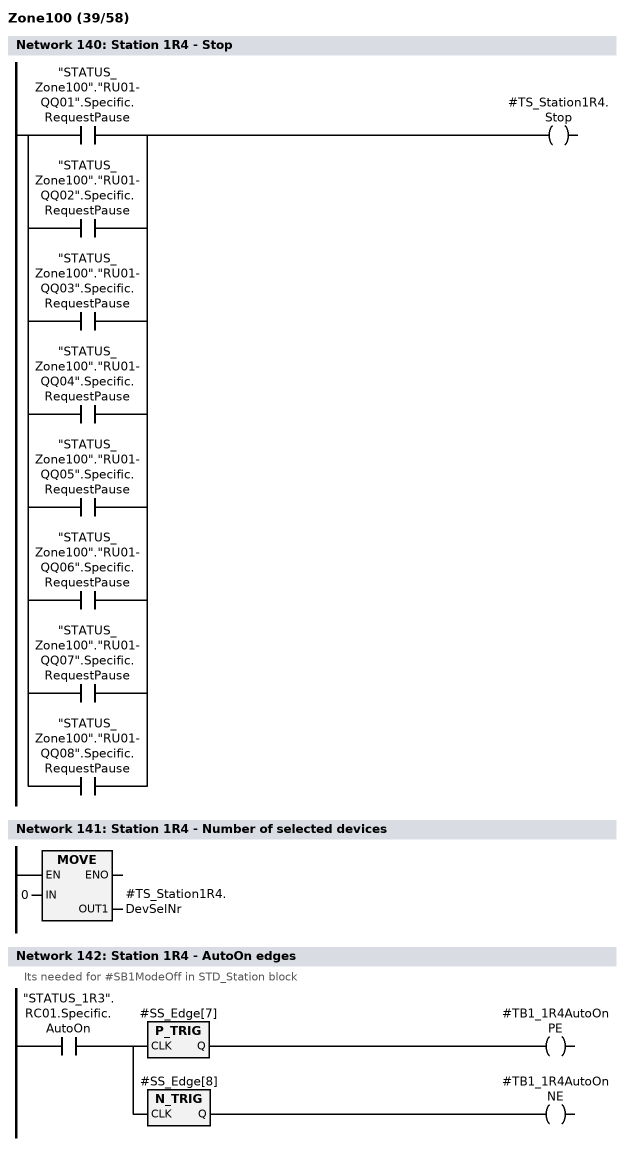
   RUNG wire#powerrail
      Contact( "STATUS_Zone100"."RU01-QQ01".Specific.RequestPause )
      wire#w1
      Coil( #TS_Station1R4.Stop )
   END_RUNG
   RUNG wire#powerrail
      Contact( "STATUS_Zone100"."RU01-QQ02".Specific.RequestPause )
   END_RUNG wire#w1
   RUNG wire#powerrail
      Contact( "STATUS_Zone100"."RU01-QQ03".Specific.RequestPause )
   END_RUNG wire#w1
   RUNG wire#powerrail
      Contact( "STATUS_Zone100"."RU01-QQ04".Specific.RequestPause )
   END_RUNG wire#w1
   RUNG wire#powerrail
      Contact( "STATUS_Zone100"."RU01-QQ05".Specific.RequestPause )
   END_RUNG wire#w1
   RUNG wire#powerrail
      Contact( "STATUS_Zone100"."RU01-QQ06".Specific.RequestPause )
   END_RUNG wire#w1
   RUNG wire#powerrail
      Contact( "STATUS_Zone100"."RU01-QQ07".Specific.RequestPause )
   END_RUNG wire#w1
   RUNG wire#powerrail
      Contact( "STATUS_Zone100"."RU01-QQ08".Specific.RequestPause )
   END_RUNG wire#w1
   // the same network as SCL:
   #TS_Station1R4.Stop := "STATUS_Zone100"."RU01-QQ01".Specific.RequestPause OR "STATUS_Zone100"."RU01-QQ02".Specific.RequestPause OR "STATUS_Zone100"."RU01-QQ03".Specific.RequestPause OR "STATUS_Zone100"."RU01-QQ04".Specific.RequestPause OR "STATUS_Zone100"."RU01-QQ05".Specific.RequestPause OR "STATUS_Zone100"."RU01-QQ06".Specific.RequestPause OR "STATUS_Zone100"."RU01-QQ07".Specific.RequestPause OR "STATUS_Zone100"."RU01-QQ08".Specific.RequestPause;
END_REGION

REGION Network 141: Station 1R4 - Number of selected devices
   RUNG wire#powerrail
      Move(in := 0, out1 => #TS_Station1R4.DevSelNr)
   END_RUNG
   // the same network as SCL:
   #TS_Station1R4.DevSelNr := 0;
END_REGION

REGION Network 142: Station 1R4 - AutoOn edges
   // Its needed for #SB1ModeOff in STD_Station block
   RUNG wire#powerrail
      Contact( "STATUS_1R3".RC01.Specific.AutoOn )
      wire#w1
      P_Trig( #SS_Edge[7] )
      Coil( #TB1_1R4AutoOnPE )
   END_RUNG
   RUNG wire#w1
      N_Trig( #SS_Edge[8] )
      Coil( #TB1_1R4AutoOnNE )
   END_RUNG
   // the same network as SCL:
   #_w1 := "STATUS_1R3".RC01.Specific.AutoOn AND NOT #SS_Edge[7];   // rising edge
   #SS_Edge[7] := "STATUS_1R3".RC01.Specific.AutoOn;
   #TB1_1R4AutoOnPE := #_w1;
   #_w2 := NOT "STATUS_1R3".RC01.Specific.AutoOn AND #SS_Edge[8];   // falling edge
   #SS_Edge[8] := "STATUS_1R3".RC01.Specific.AutoOn;
   #TB1_1R4AutoOnNE := #_w2;
END_REGION

REGION Network 143: Station 1R4 - Main control
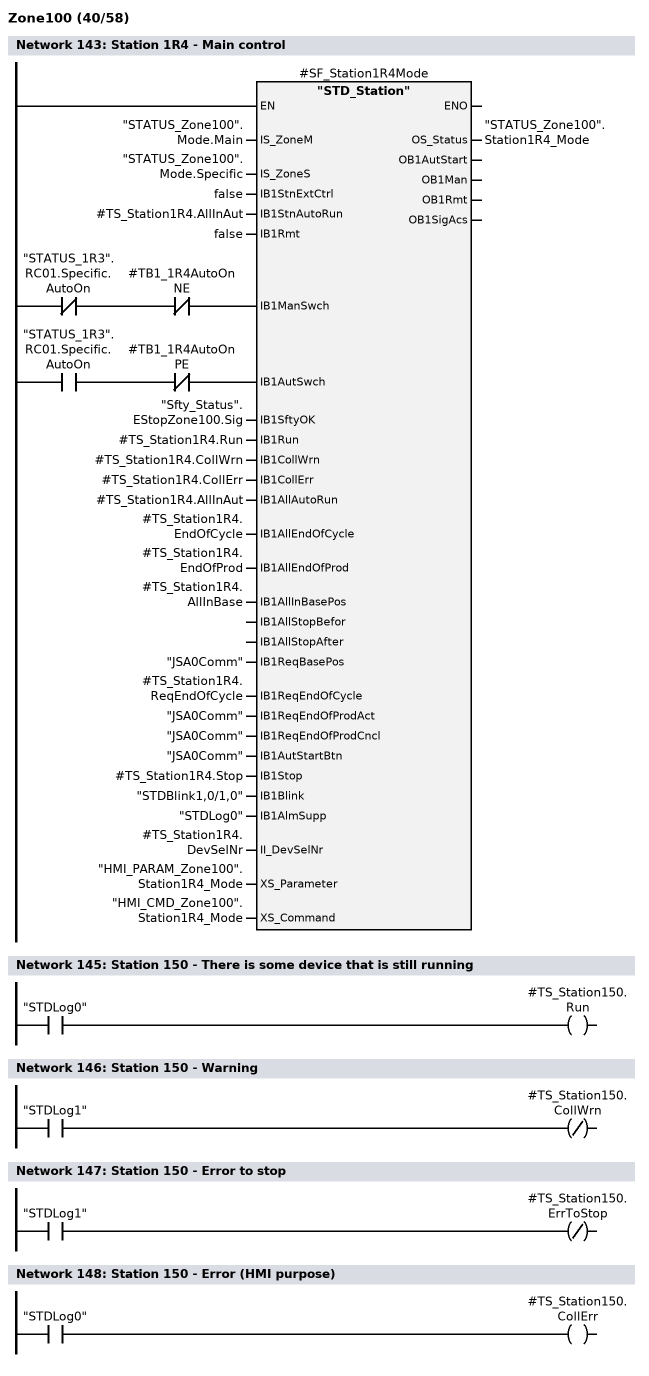
   RUNG wire#powerrail
      #SF_Station1R4Mode(IB1ManSwch := wire#w1, IB1AutSwch := wire#w2, IS_ZoneM := "STATUS_Zone100".Mode.Main, IS_ZoneS := "STATUS_Zone100".Mode.Specific, IB1StnExtCtrl := false, IB1StnAutoRun := #TS_Station1R4.AllInAut, IB1Rmt := false, IB1SftyOK := "Sfty_Status".EStopZone100.Sig, IB1Run := #TS_Station1R4.Run, IB1CollWrn := #TS_Station1R4.CollWrn, IB1CollErr := #TS_Station1R4.CollErr, IB1AllAutoRun := #TS_Station1R4.AllInAut, IB1AllEndOfCycle := #TS_Station1R4.EndOfCycle, IB1AllEndOfProd := #TS_Station1R4.EndOfProd, IB1AllInBasePos := #TS_Station1R4.AllInBase, IB1AllStopBefor :=, IB1AllStopAfter :=, IB1ReqBasePos := "JSA0Comm", IB1ReqEndOfCycle := #TS_Station1R4.ReqEndOfCycle, IB1ReqEndOfProdAct := "JSA0Comm", IB1ReqEndOfProdCncl := "JSA0Comm", IB1AutStartBtn := "JSA0Comm", IB1Stop := #TS_Station1R4.Stop, IB1Blink := "STDBlink1,0/1,0", IB1AlmSupp := "STDLog0", II_DevSelNr := #TS_Station1R4.DevSelNr, XS_Parameter := "HMI_PARAM_Zone100".Station1R4_Mode, XS_Command := "HMI_CMD_Zone100".Station1R4_Mode, OS_Status => "STATUS_Zone100".Station1R4_Mode, OB1AutStart =>, OB1Man =>, OB1Rmt =>, OB1SigAcs =>)
   END_RUNG
   RUNG wire#powerrail
      I_Contact( "STATUS_1R3".RC01.Specific.AutoOn )
      I_Contact( #TB1_1R4AutoOnNE )
   END_RUNG wire#w1
   RUNG wire#powerrail
      Contact( "STATUS_1R3".RC01.Specific.AutoOn )
      I_Contact( #TB1_1R4AutoOnPE )
   END_RUNG wire#w2
   // the same network as SCL:
   #SF_Station1R4Mode(IS_ZoneM := "STATUS_Zone100".Mode.Main,   // "STD_Station"
                      IS_ZoneS := "STATUS_Zone100".Mode.Specific,
                      IB1StnExtCtrl := false,
                      IB1StnAutoRun := #TS_Station1R4.AllInAut,
                      IB1Rmt := false,
                      IB1ManSwch := NOT "STATUS_1R3".RC01.Specific.AutoOn AND NOT #TB1_1R4AutoOnNE,
                      IB1AutSwch := "STATUS_1R3".RC01.Specific.AutoOn AND NOT #TB1_1R4AutoOnPE,
                      IB1SftyOK := "Sfty_Status".EStopZone100.Sig,
                      IB1Run := #TS_Station1R4.Run,
                      IB1CollWrn := #TS_Station1R4.CollWrn,
                      IB1CollErr := #TS_Station1R4.CollErr,
                      IB1AllAutoRun := #TS_Station1R4.AllInAut,
                      IB1AllEndOfCycle := #TS_Station1R4.EndOfCycle,
                      IB1AllEndOfProd := #TS_Station1R4.EndOfProd,
                      IB1AllInBasePos := #TS_Station1R4.AllInBase,
                      IB1ReqBasePos := "JSA0Comm",
                      IB1ReqEndOfCycle := #TS_Station1R4.ReqEndOfCycle,
                      IB1ReqEndOfProdAct := "JSA0Comm",
                      IB1ReqEndOfProdCncl := "JSA0Comm",
                      IB1AutStartBtn := "JSA0Comm",
                      IB1Stop := #TS_Station1R4.Stop,
                      IB1Blink := "STDBlink1,0/1,0",
                      IB1AlmSupp := "STDLog0",
                      II_DevSelNr := #TS_Station1R4.DevSelNr,
                      XS_Parameter := "HMI_PARAM_Zone100".Station1R4_Mode,
                      XS_Command := "HMI_CMD_Zone100".Station1R4_Mode,
                      OS_Status => "STATUS_Zone100".Station1R4_Mode);
END_REGION

REGION Network 144: *************** Station 150 ***************
END_REGION

REGION Network 145: Station 150 - There is some device that is still running
   RUNG wire#powerrail
      Contact( "STDLog0" )
      Coil( #TS_Station150.Run )
   END_RUNG
   // the same network as SCL:
   #TS_Station150.Run := "STDLog0";
END_REGION

REGION Network 146: Station 150 - Warning
   RUNG wire#powerrail
      Contact( "STDLog1" )
      I_Coil( #TS_Station150.CollWrn )
   END_RUNG
   // the same network as SCL:
   #TS_Station150.CollWrn := NOT "STDLog1";
END_REGION

REGION Network 147: Station 150 - Error to stop
   RUNG wire#powerrail
      Contact( "STDLog1" )
      I_Coil( #TS_Station150.ErrToStop )
   END_RUNG
   // the same network as SCL:
   #TS_Station150.ErrToStop := NOT "STDLog1";
END_REGION

REGION Network 148: Station 150 - Error (HMI purpose)
   RUNG wire#powerrail
      Contact( "STDLog0" )
      Coil( #TS_Station150.CollErr )
   END_RUNG
   // the same network as SCL:
   #TS_Station150.CollErr := "STDLog0";
END_REGION

REGION Network 149: Station 150 - All drives running in Automatic
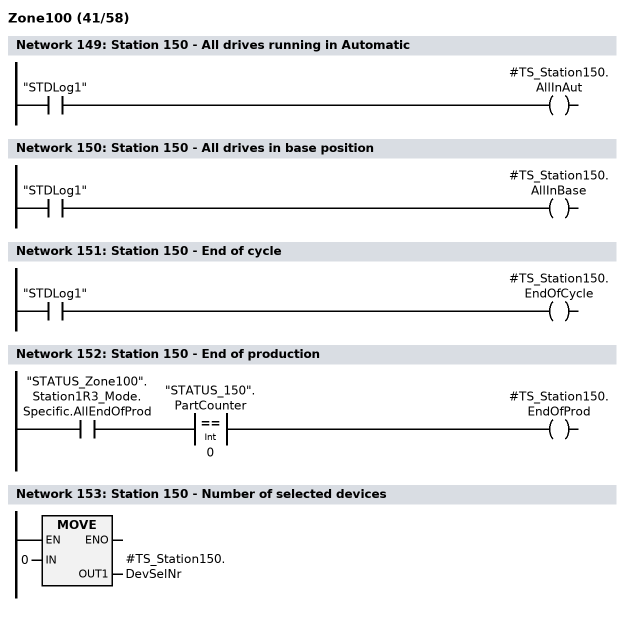
   RUNG wire#powerrail
      Contact( "STDLog1" )
      Coil( #TS_Station150.AllInAut )
   END_RUNG
   // the same network as SCL:
   #TS_Station150.AllInAut := "STDLog1";
END_REGION

REGION Network 150: Station 150 - All drives in base position
   RUNG wire#powerrail
      Contact( "STDLog1" )
      Coil( #TS_Station150.AllInBase )
   END_RUNG
   // the same network as SCL:
   #TS_Station150.AllInBase := "STDLog1";
END_REGION

REGION Network 151: Station 150 - End of cycle
   RUNG wire#powerrail
      Contact( "STDLog1" )
      Coil( #TS_Station150.EndOfCycle )
   END_RUNG
   // the same network as SCL:
   #TS_Station150.EndOfCycle := "STDLog1";
END_REGION

REGION Network 152: Station 150 - End of production
   RUNG wire#powerrail
      Contact( "STATUS_Zone100".Station1R3_Mode.Specific.AllEndOfProd )
      { S7_Templates := "SrcType := Int" } EQ_Contact(in1 := "STATUS_150".PartCounter, in2 := 0)
      Coil( #TS_Station150.EndOfProd )
   END_RUNG
   // the same network as SCL:
   #TS_Station150.EndOfProd := "STATUS_Zone100".Station1R3_Mode.Specific.AllEndOfProd AND ("STATUS_150".PartCounter = 0);
END_REGION

REGION Network 153: Station 150 - Number of selected devices
   RUNG wire#powerrail
      Move(in := 0, out1 => #TS_Station150.DevSelNr)
   END_RUNG
   // the same network as SCL:
   #TS_Station150.DevSelNr := 0;
END_REGION

REGION Network 154: Station 150 - Main control
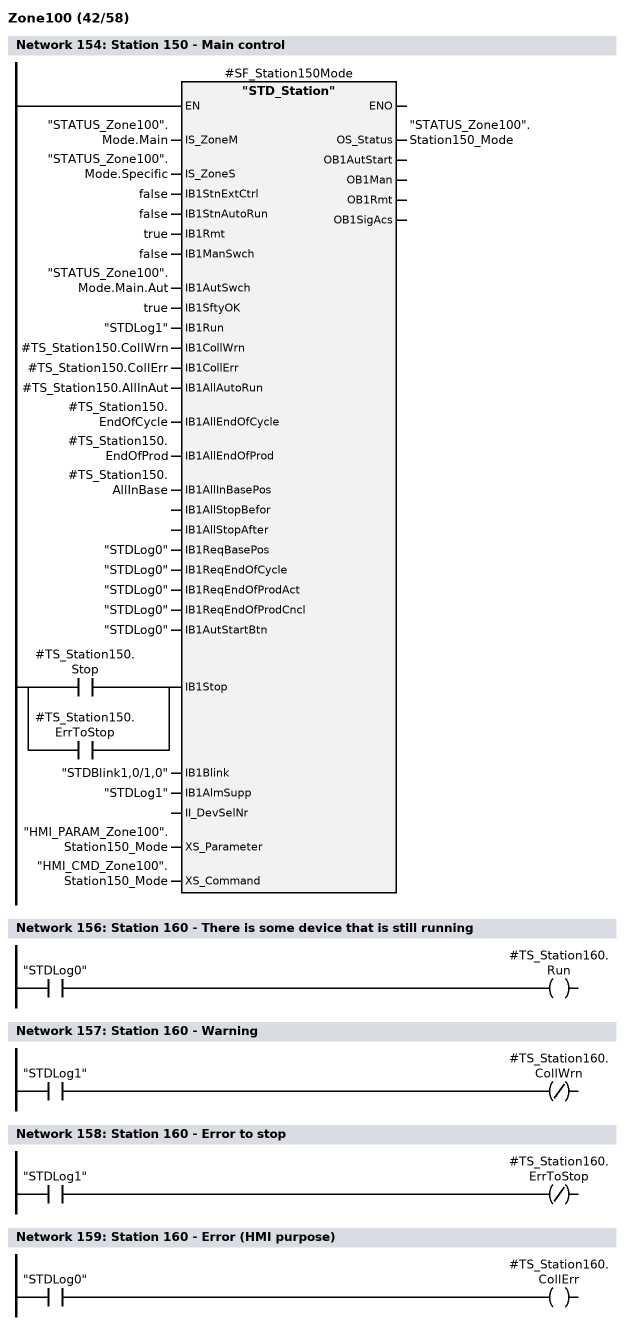
   RUNG wire#powerrail
      #SF_Station150Mode(IB1Stop := wire#w1, IS_ZoneM := "STATUS_Zone100".Mode.Main, IS_ZoneS := "STATUS_Zone100".Mode.Specific, IB1StnExtCtrl := false, IB1StnAutoRun := false, IB1Rmt := true, IB1ManSwch := false, IB1AutSwch := "STATUS_Zone100".Mode.Main.Aut, IB1SftyOK := true, IB1Run := "STDLog1", IB1CollWrn := #TS_Station150.CollWrn, IB1CollErr := #TS_Station150.CollErr, IB1AllAutoRun := #TS_Station150.AllInAut, IB1AllEndOfCycle := #TS_Station150.EndOfCycle, IB1AllEndOfProd := #TS_Station150.EndOfProd, IB1AllInBasePos := #TS_Station150.AllInBase, IB1AllStopBefor :=, IB1AllStopAfter :=, IB1ReqBasePos := "STDLog0", IB1ReqEndOfCycle := "STDLog0", IB1ReqEndOfProdAct := "STDLog0", IB1ReqEndOfProdCncl := "STDLog0", IB1AutStartBtn := "STDLog0", IB1Blink := "STDBlink1,0/1,0", IB1AlmSupp := "STDLog1", II_DevSelNr :=, XS_Parameter := "HMI_PARAM_Zone100".Station150_Mode, XS_Command := "HMI_CMD_Zone100".Station150_Mode, OS_Status => "STATUS_Zone100".Station150_Mode, OB1AutStart =>, OB1Man =>, OB1Rmt =>, OB1SigAcs =>)
   END_RUNG
   RUNG wire#powerrail
      Contact( #TS_Station150.Stop )
   END_RUNG wire#w1
   RUNG wire#powerrail
      Contact( #TS_Station150.ErrToStop )
   END_RUNG wire#w1
   // the same network as SCL:
   #SF_Station150Mode(IS_ZoneM := "STATUS_Zone100".Mode.Main,   // "STD_Station"
                      IS_ZoneS := "STATUS_Zone100".Mode.Specific,
                      IB1StnExtCtrl := false,
                      IB1StnAutoRun := false,
                      IB1Rmt := true,
                      IB1ManSwch := false,
                      IB1AutSwch := "STATUS_Zone100".Mode.Main.Aut,
                      IB1SftyOK := true,
                      IB1Run := "STDLog1",
                      IB1CollWrn := #TS_Station150.CollWrn,
                      IB1CollErr := #TS_Station150.CollErr,
                      IB1AllAutoRun := #TS_Station150.AllInAut,
                      IB1AllEndOfCycle := #TS_Station150.EndOfCycle,
                      IB1AllEndOfProd := #TS_Station150.EndOfProd,
                      IB1AllInBasePos := #TS_Station150.AllInBase,
                      IB1ReqBasePos := "STDLog0",
                      IB1ReqEndOfCycle := "STDLog0",
                      IB1ReqEndOfProdAct := "STDLog0",
                      IB1ReqEndOfProdCncl := "STDLog0",
                      IB1AutStartBtn := "STDLog0",
                      IB1Stop := #TS_Station150.Stop OR #TS_Station150.ErrToStop,
                      IB1Blink := "STDBlink1,0/1,0",
                      IB1AlmSupp := "STDLog1",
                      XS_Parameter := "HMI_PARAM_Zone100".Station150_Mode,
                      XS_Command := "HMI_CMD_Zone100".Station150_Mode,
                      OS_Status => "STATUS_Zone100".Station150_Mode);
END_REGION

REGION Network 155: *************** Station 160 ***************
END_REGION

REGION Network 156: Station 160 - There is some device that is still running
   RUNG wire#powerrail
      Contact( "STDLog0" )
      Coil( #TS_Station160.Run )
   END_RUNG
   // the same network as SCL:
   #TS_Station160.Run := "STDLog0";
END_REGION

REGION Network 157: Station 160 - Warning
   RUNG wire#powerrail
      Contact( "STDLog1" )
      I_Coil( #TS_Station160.CollWrn )
   END_RUNG
   // the same network as SCL:
   #TS_Station160.CollWrn := NOT "STDLog1";
END_REGION

REGION Network 158: Station 160 - Error to stop
   RUNG wire#powerrail
      Contact( "STDLog1" )
      I_Coil( #TS_Station160.ErrToStop )
   END_RUNG
   // the same network as SCL:
   #TS_Station160.ErrToStop := NOT "STDLog1";
END_REGION

REGION Network 159: Station 160 - Error (HMI purpose)
   RUNG wire#powerrail
      Contact( "STDLog0" )
      Coil( #TS_Station160.CollErr )
   END_RUNG
   // the same network as SCL:
   #TS_Station160.CollErr := "STDLog0";
END_REGION

REGION Network 160: Station 160 - All drives running in Automatic
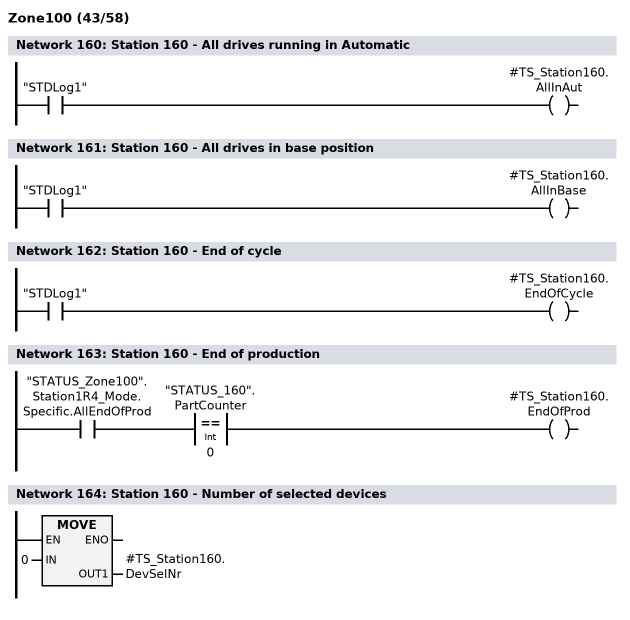
   RUNG wire#powerrail
      Contact( "STDLog1" )
      Coil( #TS_Station160.AllInAut )
   END_RUNG
   // the same network as SCL:
   #TS_Station160.AllInAut := "STDLog1";
END_REGION

REGION Network 161: Station 160 - All drives in base position
   RUNG wire#powerrail
      Contact( "STDLog1" )
      Coil( #TS_Station160.AllInBase )
   END_RUNG
   // the same network as SCL:
   #TS_Station160.AllInBase := "STDLog1";
END_REGION

REGION Network 162: Station 160 - End of cycle
   RUNG wire#powerrail
      Contact( "STDLog1" )
      Coil( #TS_Station160.EndOfCycle )
   END_RUNG
   // the same network as SCL:
   #TS_Station160.EndOfCycle := "STDLog1";
END_REGION

REGION Network 163: Station 160 - End of production
   RUNG wire#powerrail
      Contact( "STATUS_Zone100".Station1R4_Mode.Specific.AllEndOfProd )
      { S7_Templates := "SrcType := Int" } EQ_Contact(in1 := "STATUS_160".PartCounter, in2 := 0)
      Coil( #TS_Station160.EndOfProd )
   END_RUNG
   // the same network as SCL:
   #TS_Station160.EndOfProd := "STATUS_Zone100".Station1R4_Mode.Specific.AllEndOfProd AND ("STATUS_160".PartCounter = 0);
END_REGION

REGION Network 164: Station 160 - Number of selected devices
   RUNG wire#powerrail
      Move(in := 0, out1 => #TS_Station160.DevSelNr)
   END_RUNG
   // the same network as SCL:
   #TS_Station160.DevSelNr := 0;
END_REGION

REGION Network 165: Station 160 - Main control
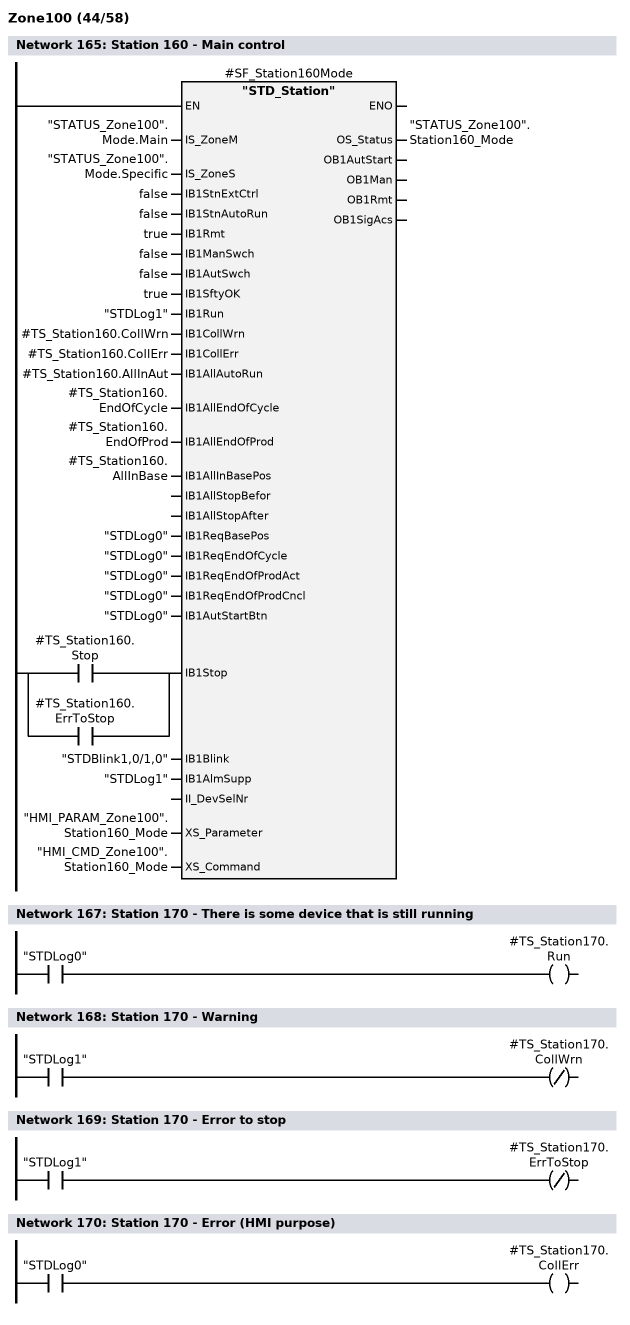
   RUNG wire#powerrail
      #SF_Station160Mode(IB1Stop := wire#w1, IS_ZoneM := "STATUS_Zone100".Mode.Main, IS_ZoneS := "STATUS_Zone100".Mode.Specific, IB1StnExtCtrl := false, IB1StnAutoRun := false, IB1Rmt := true, IB1ManSwch := false, IB1AutSwch := false, IB1SftyOK := true, IB1Run := "STDLog1", IB1CollWrn := #TS_Station160.CollWrn, IB1CollErr := #TS_Station160.CollErr, IB1AllAutoRun := #TS_Station160.AllInAut, IB1AllEndOfCycle := #TS_Station160.EndOfCycle, IB1AllEndOfProd := #TS_Station160.EndOfProd, IB1AllInBasePos := #TS_Station160.AllInBase, IB1AllStopBefor :=, IB1AllStopAfter :=, IB1ReqBasePos := "STDLog0", IB1ReqEndOfCycle := "STDLog0", IB1ReqEndOfProdAct := "STDLog0", IB1ReqEndOfProdCncl := "STDLog0", IB1AutStartBtn := "STDLog0", IB1Blink := "STDBlink1,0/1,0", IB1AlmSupp := "STDLog1", II_DevSelNr :=, XS_Parameter := "HMI_PARAM_Zone100".Station160_Mode, XS_Command := "HMI_CMD_Zone100".Station160_Mode, OS_Status => "STATUS_Zone100".Station160_Mode, OB1AutStart =>, OB1Man =>, OB1Rmt =>, OB1SigAcs =>)
   END_RUNG
   RUNG wire#powerrail
      Contact( #TS_Station160.Stop )
   END_RUNG wire#w1
   RUNG wire#powerrail
      Contact( #TS_Station160.ErrToStop )
   END_RUNG wire#w1
   // the same network as SCL:
   #SF_Station160Mode(IS_ZoneM := "STATUS_Zone100".Mode.Main,   // "STD_Station"
                      IS_ZoneS := "STATUS_Zone100".Mode.Specific,
                      IB1StnExtCtrl := false,
                      IB1StnAutoRun := false,
                      IB1Rmt := true,
                      IB1ManSwch := false,
                      IB1AutSwch := false,
                      IB1SftyOK := true,
                      IB1Run := "STDLog1",
                      IB1CollWrn := #TS_Station160.CollWrn,
                      IB1CollErr := #TS_Station160.CollErr,
                      IB1AllAutoRun := #TS_Station160.AllInAut,
                      IB1AllEndOfCycle := #TS_Station160.EndOfCycle,
                      IB1AllEndOfProd := #TS_Station160.EndOfProd,
                      IB1AllInBasePos := #TS_Station160.AllInBase,
                      IB1ReqBasePos := "STDLog0",
                      IB1ReqEndOfCycle := "STDLog0",
                      IB1ReqEndOfProdAct := "STDLog0",
                      IB1ReqEndOfProdCncl := "STDLog0",
                      IB1AutStartBtn := "STDLog0",
                      IB1Stop := #TS_Station160.Stop OR #TS_Station160.ErrToStop,
                      IB1Blink := "STDBlink1,0/1,0",
                      IB1AlmSupp := "STDLog1",
                      XS_Parameter := "HMI_PARAM_Zone100".Station160_Mode,
                      XS_Command := "HMI_CMD_Zone100".Station160_Mode,
                      OS_Status => "STATUS_Zone100".Station160_Mode);
END_REGION

REGION Network 166: *************** Station 170 ***************
END_REGION

REGION Network 167: Station 170 - There is some device that is still running
   RUNG wire#powerrail
      Contact( "STDLog0" )
      Coil( #TS_Station170.Run )
   END_RUNG
   // the same network as SCL:
   #TS_Station170.Run := "STDLog0";
END_REGION

REGION Network 168: Station 170 - Warning
   RUNG wire#powerrail
      Contact( "STDLog1" )
      I_Coil( #TS_Station170.CollWrn )
   END_RUNG
   // the same network as SCL:
   #TS_Station170.CollWrn := NOT "STDLog1";
END_REGION

REGION Network 169: Station 170 - Error to stop
   RUNG wire#powerrail
      Contact( "STDLog1" )
      I_Coil( #TS_Station170.ErrToStop )
   END_RUNG
   // the same network as SCL:
   #TS_Station170.ErrToStop := NOT "STDLog1";
END_REGION

REGION Network 170: Station 170 - Error (HMI purpose)
   RUNG wire#powerrail
      Contact( "STDLog0" )
      Coil( #TS_Station170.CollErr )
   END_RUNG
   // the same network as SCL:
   #TS_Station170.CollErr := "STDLog0";
END_REGION

REGION Network 171: Station 170 - All drives running in Automatic
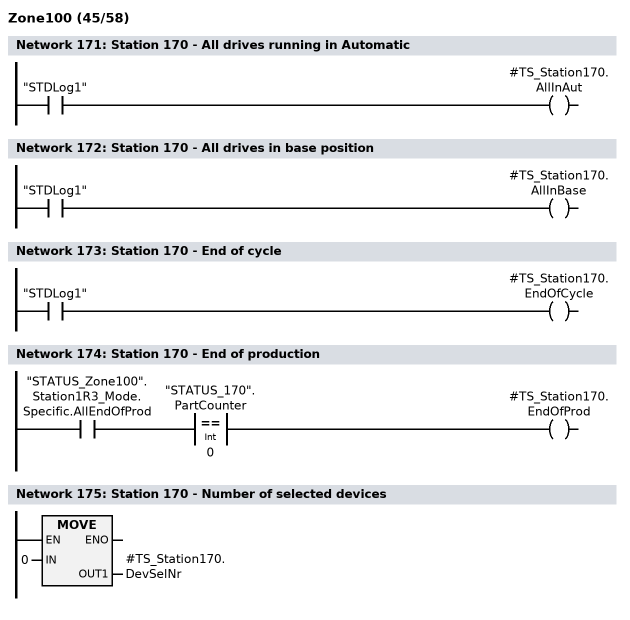
   RUNG wire#powerrail
      Contact( "STDLog1" )
      Coil( #TS_Station170.AllInAut )
   END_RUNG
   // the same network as SCL:
   #TS_Station170.AllInAut := "STDLog1";
END_REGION

REGION Network 172: Station 170 - All drives in base position
   RUNG wire#powerrail
      Contact( "STDLog1" )
      Coil( #TS_Station170.AllInBase )
   END_RUNG
   // the same network as SCL:
   #TS_Station170.AllInBase := "STDLog1";
END_REGION

REGION Network 173: Station 170 - End of cycle
   RUNG wire#powerrail
      Contact( "STDLog1" )
      Coil( #TS_Station170.EndOfCycle )
   END_RUNG
   // the same network as SCL:
   #TS_Station170.EndOfCycle := "STDLog1";
END_REGION

REGION Network 174: Station 170 - End of production
   RUNG wire#powerrail
      Contact( "STATUS_Zone100".Station1R3_Mode.Specific.AllEndOfProd )
      { S7_Templates := "SrcType := Int" } EQ_Contact(in1 := "STATUS_170".PartCounter, in2 := 0)
      Coil( #TS_Station170.EndOfProd )
   END_RUNG
   // the same network as SCL:
   #TS_Station170.EndOfProd := "STATUS_Zone100".Station1R3_Mode.Specific.AllEndOfProd AND ("STATUS_170".PartCounter = 0);
END_REGION

REGION Network 175: Station 170 - Number of selected devices
   RUNG wire#powerrail
      Move(in := 0, out1 => #TS_Station170.DevSelNr)
   END_RUNG
   // the same network as SCL:
   #TS_Station170.DevSelNr := 0;
END_REGION

REGION Network 176: Station 170 - Main control
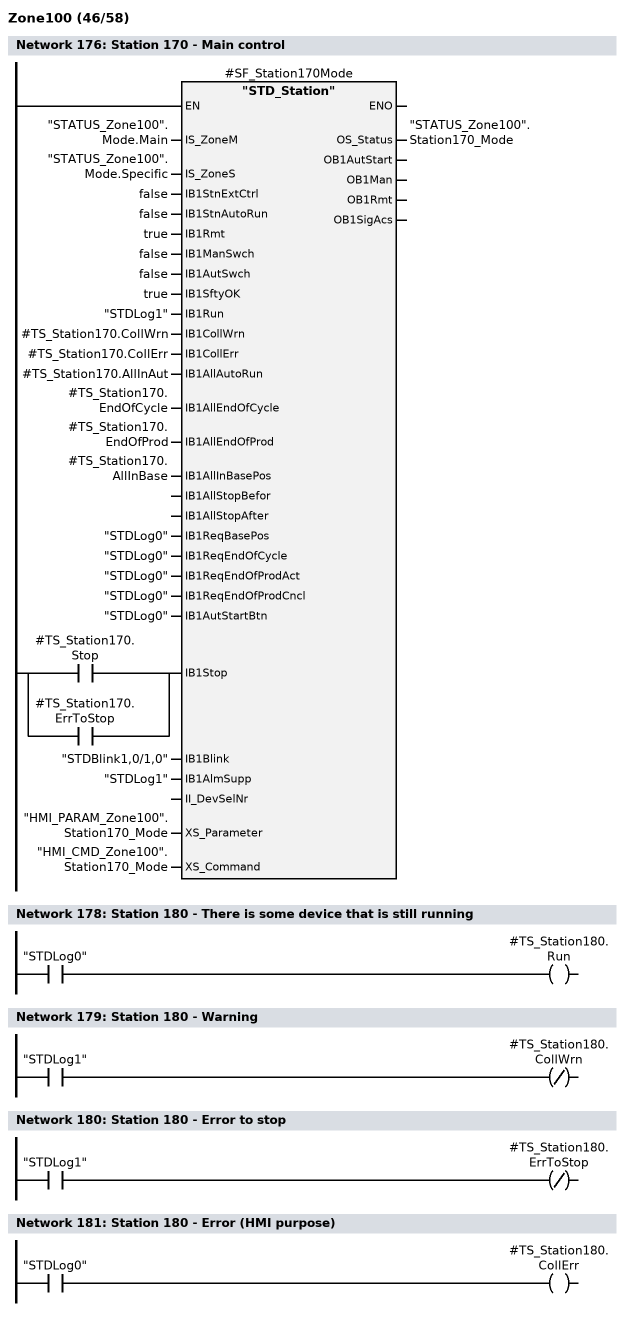
   RUNG wire#powerrail
      #SF_Station170Mode(IB1Stop := wire#w1, IS_ZoneM := "STATUS_Zone100".Mode.Main, IS_ZoneS := "STATUS_Zone100".Mode.Specific, IB1StnExtCtrl := false, IB1StnAutoRun := false, IB1Rmt := true, IB1ManSwch := false, IB1AutSwch := false, IB1SftyOK := true, IB1Run := "STDLog1", IB1CollWrn := #TS_Station170.CollWrn, IB1CollErr := #TS_Station170.CollErr, IB1AllAutoRun := #TS_Station170.AllInAut, IB1AllEndOfCycle := #TS_Station170.EndOfCycle, IB1AllEndOfProd := #TS_Station170.EndOfProd, IB1AllInBasePos := #TS_Station170.AllInBase, IB1AllStopBefor :=, IB1AllStopAfter :=, IB1ReqBasePos := "STDLog0", IB1ReqEndOfCycle := "STDLog0", IB1ReqEndOfProdAct := "STDLog0", IB1ReqEndOfProdCncl := "STDLog0", IB1AutStartBtn := "STDLog0", IB1Blink := "STDBlink1,0/1,0", IB1AlmSupp := "STDLog1", II_DevSelNr :=, XS_Parameter := "HMI_PARAM_Zone100".Station170_Mode, XS_Command := "HMI_CMD_Zone100".Station170_Mode, OS_Status => "STATUS_Zone100".Station170_Mode, OB1AutStart =>, OB1Man =>, OB1Rmt =>, OB1SigAcs =>)
   END_RUNG
   RUNG wire#powerrail
      Contact( #TS_Station170.Stop )
   END_RUNG wire#w1
   RUNG wire#powerrail
      Contact( #TS_Station170.ErrToStop )
   END_RUNG wire#w1
   // the same network as SCL:
   #SF_Station170Mode(IS_ZoneM := "STATUS_Zone100".Mode.Main,   // "STD_Station"
                      IS_ZoneS := "STATUS_Zone100".Mode.Specific,
                      IB1StnExtCtrl := false,
                      IB1StnAutoRun := false,
                      IB1Rmt := true,
                      IB1ManSwch := false,
                      IB1AutSwch := false,
                      IB1SftyOK := true,
                      IB1Run := "STDLog1",
                      IB1CollWrn := #TS_Station170.CollWrn,
                      IB1CollErr := #TS_Station170.CollErr,
                      IB1AllAutoRun := #TS_Station170.AllInAut,
                      IB1AllEndOfCycle := #TS_Station170.EndOfCycle,
                      IB1AllEndOfProd := #TS_Station170.EndOfProd,
                      IB1AllInBasePos := #TS_Station170.AllInBase,
                      IB1ReqBasePos := "STDLog0",
                      IB1ReqEndOfCycle := "STDLog0",
                      IB1ReqEndOfProdAct := "STDLog0",
                      IB1ReqEndOfProdCncl := "STDLog0",
                      IB1AutStartBtn := "STDLog0",
                      IB1Stop := #TS_Station170.Stop OR #TS_Station170.ErrToStop,
                      IB1Blink := "STDBlink1,0/1,0",
                      IB1AlmSupp := "STDLog1",
                      XS_Parameter := "HMI_PARAM_Zone100".Station170_Mode,
                      XS_Command := "HMI_CMD_Zone100".Station170_Mode,
                      OS_Status => "STATUS_Zone100".Station170_Mode);
END_REGION

REGION Network 177: *************** Station 180 ***************
END_REGION

REGION Network 178: Station 180 - There is some device that is still running
   RUNG wire#powerrail
      Contact( "STDLog0" )
      Coil( #TS_Station180.Run )
   END_RUNG
   // the same network as SCL:
   #TS_Station180.Run := "STDLog0";
END_REGION

REGION Network 179: Station 180 - Warning
   RUNG wire#powerrail
      Contact( "STDLog1" )
      I_Coil( #TS_Station180.CollWrn )
   END_RUNG
   // the same network as SCL:
   #TS_Station180.CollWrn := NOT "STDLog1";
END_REGION

REGION Network 180: Station 180 - Error to stop
   RUNG wire#powerrail
      Contact( "STDLog1" )
      I_Coil( #TS_Station180.ErrToStop )
   END_RUNG
   // the same network as SCL:
   #TS_Station180.ErrToStop := NOT "STDLog1";
END_REGION

REGION Network 181: Station 180 - Error (HMI purpose)
   RUNG wire#powerrail
      Contact( "STDLog0" )
      Coil( #TS_Station180.CollErr )
   END_RUNG
   // the same network as SCL:
   #TS_Station180.CollErr := "STDLog0";
END_REGION

REGION Network 182: Station 180 - All drives running in Automatic
